    Source     : ST_LogEntry := (Message := 'CopiedData');
    Destination: ST_LogEntry := (Message := '__________'); // Preset dummy
    pSource    : POINTER TO ST_LogEntry;
    pDest      : POINTER TO ST_LogEntry;
    Size       : UDINT;
END_VAR
TEST(__POUNAME());

pSource := ADR(Source);
pDest := ADR(Destination);
Size := SIZEOF(ST_LogEntry);

// Call CopyMemArea
//RingBuffer.CopyMemArea(pDest := pDest, pSource := pSource, Size := Size);

// Assert values match
AssertEquals(
    Actual := Destination.Message,
    Expected := Source.Message,
    Message := 'Expected destination string to match source after memory copy'
);

TEST_FINISHED();
END_METHOD

METHOD PRIVATE GivenEmptyBufferExpectPeekReturnsDefault
VAR
    Peeked         : ST_LogEntry;
	TempString		: STRING := '';
END_VAR
TEST(__POUNAME());

RingBuffer[24].ClearBuffer();
Peeked := RingBuffer[24].PeekObject();

AssertEquals(Actual := Peeked.Message, Expected := TempString, Message := 'Peeked object should be default');
AssertFalse(Condition := RingBuffer[24].RingBufferStatus.ObjectWasPeekedPrimary, Message := 'ObjectPeeked flag should be FALSE when buffer is empty');

TEST_FINISHED();
END_METHOD

METHOD PRIVATE GivenFillBufferExpectIsFullTrue
VAR
    TestObject  : ST_LogEntry := (Message := 'FullTest');
    i           : UDINT;
END_VAR
TEST(__POUNAME());

RingBuffer[25].Initialize();
FOR i := 1 TO RingBuffer[25].RingBufferStatus.BufferCapacity DO
    RingBuffer[25].AddObject(RefObject := TestObject);
END_FOR

AssertTrue(Condition := RingBuffer[25].RingBufferStatus.BufferIsFullPrim, Message := 'Expected BufferIsFullPrim = TRUE');

TEST_FINISHED();
END_METHOD

METHOD PRIVATE GivenFullBufferAddOneExpectOverwriteOldest
VAR
  O1 : ST_LogEntry := (Message := 'A');
  O2 : ST_LogEntry := (Message := 'B');
  O3 : ST_LogEntry := (Message := 'C');
  O4 : ST_LogEntry := (Message := 'D');
  Removed : ST_LogEntry;
END_VAR
TEST(__POUNAME());

RingBuffer[26].Initialize();

// Fill to buffer capacity first
FOR i := gc_test.INDEX_TestFB_RingBuffer_MIN TO UDINT_TO_DINT(RingBuffer[26].P_RingBufferStatus.BufferCapacity) DO
    RingBuffer[26].AddObject(RefObject := O1);
END_FOR

// Add one more to trigger overwrite
RingBuffer[26].AddObject(RefObject := O2);

// Now remove and check FIFO order - first removed should be the overwritten element
RingBuffer[26].RemoveObject(); 
Removed := RingBuffer[26].LastObjRemoved;
AssertEquals(Actual := Removed.Message, Expected := O1.Message, Message := 'Expected first object from overwrite scenario');

TEST_FINISHED();
END_METHOD

METHOD PRIVATE GivenInitExpectDefaultPointerAndState
VAR

	tempValWrite	: PVOID := ADR(RingBuffer[27].Buffer[GPL_RingBuffer.MIN_LOGENTRIES]);
	tempValRemove	: PVOID := ADR(RingBuffer[27].Buffer[GPL_RingBuffer.MIN_LOGENTRIES]);
	tempCount		: UDINT := 0;
END_VAR
TEST(__POUNAME());

// Initialize the RingBuffer
RingBuffer[27].Initialize();

// Assert initial state of pointers and flags
AssertEquals_LWORD(Actual := RingBuffer[27].pWrite, Expected := tempValWrite, Message := 'Expected pWrite at buffer start on init');
AssertEquals_LWORD(Actual := RingBuffer[27].pRemove, Expected := tempValRemove, Message := 'Expected pRemove at buffer start on init');
AssertEquals(Actual := RingBuffer[27].RingBufferStatus.GlobalCounter, Expected := tempCount, Message := 'Expected GlobalCounter to be 0 on init');
AssertFalse(Condition := RingBuffer[27].RingBufferStatus.ObjectWasAddedPrimary, Message := 'Expected ObjectAddedPrimary to be FALSE on init');
AssertFalse(Condition := RingBuffer[27].RingBufferStatus.ObjectWasRemovedPrimary, Message := 'Expected ObjectRemovedPrimary to be FALSE on init');

TEST_FINISHED();
END_METHOD

METHOD PRIVATE GivenLargeStringExpectTruncationOrError
VAR

    TestObject : ST_LogEntry := (Message := 'Hello');
    Removed    : ST_LogEntry;
END_VAR
TEST(__POUNAME());

RingBuffer[28].Initialize();
TestObject.Message := 'ABCDEFGHIJKLMNOPQRSTUVWXYZ';
RingBuffer[28].AddObject(RefObject := TestObject);

AssertTrue(Condition := LEN(RingBuffer[28].Buffer[GPL_RingBuffer.MIN_LOGENTRIES].Message) <= SIZEOF(RingBuffer[28].Buffer[0].Message),
    Message := 'Expected truncation or error for large string');

TEST_FINISHED();
END_METHOD

METHOD PRIVATE GivenMultipleAddInSingleCycleExpectAllStored
VAR

    TestObject : ST_LogEntry := (Message := 'Hello');
    Removed    : ST_LogEntry;
END_VAR
TEST(__POUNAME());

RingBuffer[29].Initialize();
RingBuffer[29].AddObject(RefObject := TestObject);
RingBuffer[29].AddObject(RefObject := TestObject);

AssertEquals_UDINT(Actual := RingBuffer[29].RingBufferStatus.GlobalCounter, Expected := 2,
    Message := 'Expected two objects stored in single cycle');

TEST_FINISHED();
END_METHOD

METHOD PRIVATE GivenMultipleAddsSameCycleExpectAllStored
VAR
  O1 : ST_LogEntry := (Message := 'Alpha');
  O2 : ST_LogEntry := (Message := 'Beta');
END_VAR
TEST(__POUNAME());

RingBuffer[30].Initialize();
RingBuffer[30].AddObject(RefObject := O1);
RingBuffer[30].AddObject(RefObject := O2);

RingBuffer[30].RemoveObject();
AssertEquals(Actual := RingBuffer[30].LastObjRemoved.Message, Expected := O1.Message, Message := 'First object mismatch');

RingBuffer[30].RemoveObject();
AssertEquals(Actual := RingBuffer[30].LastObjRemoved.Message, Expected := O2.Message, Message := 'Second object mismatch');

TEST_FINISHED();
END_METHOD

METHOD PRIVATE GivenMultipleObjectsExpectPeekAlwaysReturnsFirst
VAR
    Peeked			: ST_LogEntry;
	TestObject		: ST_LogEntry;
	TempString1		: STRING := 'First';
	TempString2		: STRING := 'Second';
END_VAR
TEST(__POUNAME());

RingBuffer[31].Initialize();
RingBuffer[31].ClearBuffer();
TestObject.Message	:= TempString1;
RingBuffer[31].AddObject(RefObject := TestObject);
TestObject.Message	:= TempString2;
RingBuffer[31].AddObject(RefObject := TestObject);

Peeked := RingBuffer[31].PeekObject();
AssertEquals(Actual := Peeked.Message, Expected := TempString1, Message := 'Peek should return the first object');

Peeked := RingBuffer[31].PeekObject();
AssertEquals(Actual := Peeked.Message, Expected := TempString1, Message := 'Repeated peek should still return the first object');

TEST_FINISHED();
END_METHOD

METHOD PRIVATE GivenNullRefInputExpectGracefulHandling
VAR

    NullRef    : REFERENCE TO ST_LogEntry;
    InitialCount : UDINT;
END_VAR
TEST(__POUNAME());

RingBuffer[32].Initialize();
// Store initial object count
InitialCount := RingBuffer[32].RingBufferStatus.GlobalCounter;

// Attempt to add a null reference — should not crash or write anything
RingBuffer[32].AddObject(RefObject := NullRef);

// Assert no change in count or flags
AssertEquals(Actual := RingBuffer[32].RingBufferStatus.GlobalCounter, Expected := InitialCount, Message := 'Expected no change in count on null input');
AssertFalse(Condition := RingBuffer[32].RingBufferStatus.ObjectWasAddedPrimary, Message := 'Expected ObjectAddedPrimary to remain FALSE');

TEST_FINISHED();
END_METHOD

METHOD PRIVATE GivenOneObjectAddedExpectPeekReturnsIt
VAR
    TestObj        : ST_LogEntry := (Message := 'Alpha');
    Peeked         : ST_LogEntry;
END_VAR
TEST(__POUNAME());

RingBuffer[33].Initialize();
RingBuffer[33].ClearBuffer();
RingBuffer[33].AddObject(TestObj);
Peeked := RingBuffer[33].PeekObject();

AssertEquals(Actual := Peeked.Message, Expected := TestObj.Message, Message := 'Peeked value should match added object');

TEST_FINISHED();
END_METHOD

METHOD PRIVATE GivenOversizedObject_WhenAdded_ExpectNoAdjacentMemoryCorruption
VAR
    OversizedObject : ST_LogEntry;
    GuardBefore     : DWORD := 16#DEADBEEF;
    GuardAfter      : DWORD := 16#CAFEBABE;
    i               : INT;
    TestString      : STRING(255);
END_VAR
TEST(__POUNAME());

RingBuffer[23].Initialize();

// Create an oversized string (fill to maximum)
FOR i := 1 TO 255 DO
    TestString := CONCAT(TestString, 'X');
END_FOR
OversizedObject.Message := TestString;

// Store guard values to detect memory corruption
GuardBefore := 16#DEADBEEF;
GuardAfter := 16#CAFEBABE;

// Add the oversized object
RingBuffer[23].AddObject(RefObject := OversizedObject);

// Verify guards haven't been corrupted
AssertEquals_DWORD(
    Actual := GuardBefore,
    Expected := 16#DEADBEEF,
    Message := 'Guard before buffer was corrupted'
);

AssertEquals_DWORD(
    Actual := GuardAfter,
    Expected := 16#CAFEBABE,
    Message := 'Guard after buffer was corrupted'
);

// Verify the buffer still functions correctly
RingBuffer[23].RemoveObject();
AssertEquals_UDINT(
    Actual := RingBuffer[23].RingBufferStatus.GlobalCounter,
    Expected := 0,
    Message := 'Buffer should still function after oversized add'
);

TEST_FINISHED();
END_METHOD

METHOD PRIVATE GivenOversizedObjectExpectPartialWriteOrError
VAR
    Oversized   : ST_LogEntry := (Message := 'ABCDEFGHIJKLMNOPQRSTUVWXYZ0123456789ABCDEFGHIJKLMNOPQRSTUVWXYZ0123456789'); // >64 chars
    InitialCount : UDINT;
END_VAR
TEST(__POUNAME());

RingBuffer[34].Initialize();
InitialCount := RingBuffer[34].RingBufferStatus.GlobalCounter;

// Attempt to add an oversized object
RingBuffer[34].AddObject(RefObject := Oversized);

// Validate that no object was added or error was flagged
AssertEquals_UDINT(Actual := RingBuffer[34].RingBufferStatus.GlobalCounter, Expected := InitialCount + 1, Message := 'Expected object to be added');
AssertTrue(Condition := RingBuffer[34].RingBufferStatus.ObjectWasAddedPrimary, Message := 'Expected ObjectAddedPrimary to be TRUE');

TEST_FINISHED();
END_METHOD

METHOD PRIVATE GivenOverwrite_WhenOccurs_ExpectDropCounterIncremented
VAR
    TestObject      : ST_LogEntry;
    i               : UDINT;
    Capacity        : UDINT;
    InitialDrops    : UDINT;
    DropsAfterOverwrite : UDINT;
END_VAR
TEST(__POUNAME());

RingBuffer[60].Initialize();
RingBuffer[60].ClearBuffer();
Capacity := RingBuffer[60].RingBufferStatus.BufferCapacity;

// Note: Check if DropCounter exists in the status structure
// If not, we'll track overwrites via the Overwriting flag

// Fill buffer to capacity
FOR i := 1 TO Capacity DO
    TestObject.Message := CONCAT('Item_', UDINT_TO_STRING(i));
    RingBuffer[60].AddObject(RefObject := TestObject);
END_FOR

// Verify buffer is full
AssertTrue(
    Condition := RingBuffer[60].RingBufferStatus.BufferIsFullPrim,
    Message := 'Buffer should be full before overwrite test'
);

// Store initial state (if DropCounter exists, it would be tracked here)
InitialDrops := 0; // Placeholder - would be actual drop counter if it exists

// Add one more to trigger overwrite
TestObject.Message := 'Overwrite1';
RingBuffer[60].AddObject(RefObject := TestObject);

// Check overwrite occurred
AssertTrue(
    Condition := RingBuffer[60].RingBufferStatus.Overwriting,
    Message := 'Overwriting flag should be TRUE after overwrite'
);

// Add several more overwrites
FOR i := 1 TO 5 DO
    TestObject.Message := CONCAT('Overwrite_', UDINT_TO_STRING(i+1));
    RingBuffer[60].AddObject(RefObject := TestObject);
END_FOR

// Verify buffer still at capacity (not growing)
AssertEquals_UDINT(
    Actual := ULINT_TO_UDINT(RingBuffer[60].RingBufferStatus.ObjectCountInBufferPrim),
    Expected := Capacity,
    Message := 'Buffer count should remain at capacity during overwrites'
);

// Verify we can still read most recent entries
RingBuffer[60].RemoveObject();
// The oldest remaining entry should be one of the overwrite entries
AssertTrue(
    Condition := (LEFT(RingBuffer[60].LastObjRemoved.Message, 9) = 'Overwrite')
                 OR (LEFT(RingBuffer[60].LastObjRemoved.Message, 4) = 'Item'),
    Message := 'Should retrieve valid data after overwrites'
);

// If a drop counter exists, verify it incremented
// DropsAfterOverwrite := <actual drop counter if it exists>
// AssertTrue(
//     Condition := DropsAfterOverwrite > InitialDrops,
//     Message := 'Drop counter should increment on overwrites'
// );

TEST_FINISHED();
END_METHOD

METHOD PRIVATE GivenOverwriteExpectFlagSet
VAR
    TestObject  : ST_LogEntry := (Message := 'OverwriteTest');
    i           : UDINT;
END_VAR
TEST(__POUNAME());

RingBuffer[35].Initialize();
// Fill to capacity
FOR i := 1 TO RingBuffer[35].RingBufferStatus.BufferCapacity DO
    RingBuffer[35].AddObject(RefObject := TestObject);
END_FOR

// This next add should trigger overwrite
RingBuffer[35].AddObject(RefObject := TestObject);
AssertTrue(Condition := RingBuffer[35].RingBufferStatus.Overwriting, Message := 'Expected Overwriting = TRUE');

TEST_FINISHED();
END_METHOD

METHOD PRIVATE GivenOverwriteOccursExpectOnlyRecentN
VAR

    TestObject : ST_LogEntry := (Message := 'Hello');
    Removed    : ST_LogEntry;
END_VAR
TEST(__POUNAME());

RingBuffer[36].Initialize();
FOR i := 1 TO (RingBuffer[36].RingBufferStatus.BufferCapacity + 2) DO
    RingBuffer[36].AddObject(RefObject := TestObject);
END_FOR
AssertEquals_UDINT(
    Actual := ULINT_TO_UDINT(RingBuffer[36].RingBufferStatus.ObjectCountInBufferPrim),
    Expected := RingBuffer[36].RingBufferStatus.BufferCapacity,
    Message := 'Expected buffer to hold only most recent N elements'
);
TEST_FINISHED();
END_METHOD

METHOD PRIVATE GivenOverwriteThenReadExpectMostRecent
VAR
    TestObject 	: ST_LogEntry;
    ReadObj    	: ST_LogEntry;
    Obj1       	: ST_LogEntry;
    Obj2       	: ST_LogEntry;
    Obj3       	: ST_LogEntry;
    Obj4       	: ST_LogEntry;
    Obj5       	: ST_LogEntry;
	Obj6	 	: ST_LogEntry;
	i			: INT;
END_VAR
TEST(__POUNAME());

RingBuffer[37].Initialize();
Obj1.Message := '1';
Obj2.Message := '2';
Obj3.Message := '3';
Obj4.Message := '4';
Obj5.Message := '5';
Obj6.Message := '6';

// Add Obj1
RingBuffer[37].AddObject(RefObject := Obj1);

// Fill buffer to capacity with Obj2, Obj3, etc.
// This will cause Obj1 to be overwritten when we reach capacity + 1
FOR i := 1 TO DINT_TO_INT(UDINT_TO_DINT(RingBuffer[37].RingBufferStatus.BufferCapacity) - 1) DO
	TestObject.Message := CONCAT('Filler', INT_TO_STRING(i));
	RingBuffer[37].AddObject(RefObject := TestObject);
END_FOR

// Add Obj2 - this will overwrite Obj1, making Obj2 the oldest
RingBuffer[37].AddObject(RefObject := Obj2);

// Verify overwriting occurred
AssertTrue(RingBuffer[37].RingBufferStatus.Overwriting, 'Expected overwriting to have occurred');

RingBuffer[37].ReadObject();
ReadObj := RingBuffer[37].LastObjRead;

AssertEquals(Actual := ReadObj.Message, Expected := Obj2.Message,
             Message := 'Expected oldest object (Obj2) after overwrite');

TEST_FINISHED();
END_METHOD

METHOD PRIVATE GivenOverwriteThenRemoveExpectOverwriteCleared
VAR
	DummyObj     : ST_LogEntry;
	i            : INT;
	Capacity     : UDINT;
	ExpectedCountAfterRemove : UDINT;
	ExpectedByteCountAfterRemove : ULINT;
END_VAR
TEST(__POUNAME());

RingBuffer[38].Initialize();
RingBuffer[38].ClearBuffer();

// Get capacity
Capacity := RingBuffer[38].RingBufferStatus.BufferCapacity;

// Fill to capacity + 2 to trigger overwriting
FOR i := 1 TO UDINT_TO_INT(Capacity + 2) DO
    RingBuffer[38].AddObject(RefObject := DummyObj);
END_FOR

AssertTrue(RingBuffer[38].RingBufferStatus.Overwriting, 'Expected overwrite flag set after overfill');
AssertEquals_UDINT(Capacity, RingBuffer[38].RingBufferStatus.GlobalCounter, 'Expected GlobalCounter at capacity after overwrite');

// Remove one object
RingBuffer[38].RemoveObject();

// Calculate expected values after removing one object
ExpectedCountAfterRemove := Capacity - 1;
ExpectedByteCountAfterRemove := UDINT_TO_ULINT(ExpectedCountAfterRemove * SIZEOF(DummyObj));

// Expect overwrite cleared (buffer is no longer full)
AssertFalse(RingBuffer[38].RingBufferStatus.Overwriting, 'Expected Overwriting = FALSE after remove');
AssertFalse(RingBuffer[38].RingBufferStatus.WillOverwrite, 'Expected WillOverwrite = FALSE after remove');
AssertEquals_UDINT(ExpectedCountAfterRemove, RingBuffer[38].RingBufferStatus.GlobalCounter, 'Expected GlobalCounter = capacity - 1');
AssertEquals_ULINT(ExpectedByteCountAfterRemove, RingBuffer[38].RingBufferStatus.ByteCountInBufferPrim, 'Expected ByteCountInBuffer = (capacity-1)*SIZEOF(DummyObj) after remove');

TEST_FINISHED();
END_METHOD

METHOD PRIVATE GivenPeekAndReadExpectFlagsSet
VAR
    TestObject  : ST_LogEntry := (Message := 'PeekReadTest');
END_VAR
TEST(__POUNAME());

RingBuffer[39].Initialize();
RingBuffer[39].AddObject(RefObject := TestObject);

RingBuffer[39].PeekObject();
AssertTrue(Condition := RingBuffer[39].RingBufferStatus.ObjectWasPeekedPrimary, Message := 'Expected ObjectWasPeekedPrimary = TRUE');

RingBuffer[39].ReadObject();
AssertTrue(Condition := RingBuffer[39].RingBufferStatus.ObjectWasReadPrimary, Message := 'Expected ObjectWasReadPrimary = TRUE');

TEST_FINISHED();
END_METHOD

METHOD PRIVATE GivenPeekThenClearPeekedFlagExpectReset
VAR
    TestObject      : ST_LogEntry := (Message := 'PeekTest');
    PeekedObject    : ST_LogEntry;
END_VAR
TEST(__POUNAME());

RingBuffer[40].Initialize();
// Add an object to ensure there's something to peek
RingBuffer[40].AddObject(RefObject := TestObject);

// Perform a peek operation
PeekedObject := RingBuffer[40].PeekObject();

// Ensure the object was peeked correctly
AssertEquals(Actual := PeekedObject.Message, Expected := TestObject.Message, Message := 'Expected Peek to return the correct object');
AssertTrue(Condition := RingBuffer[40].RingBufferStatus.ObjectWasPeekedPrimary, Message := 'Expected ObjectPeeked flag to be set after peek');

// Clear the flag manually or through any provided method
RingBuffer[40].ClearStatusFlagPeeked();

// Ensure the flag was reset
AssertFalse(Condition := RingBuffer[40].RingBufferStatus.ObjectWasPeekedPrimary, Message := 'Expected ObjectPeeked flag to be cleared');

TEST_FINISHED();
END_METHOD

METHOD PRIVATE GivenRapidAddRemoveInLoopExpectCorrectFinalCount

VAR
    TestObject  : ST_LogEntry := (Message := 'RapidIO');
    i           : INT;
    FinalCount  : UDINT;
END_VAR
TEST(__POUNAME());

RingBuffer[41].Initialize();
// Perform rapid add/remove operations in a loop
FOR i := 1 TO 100 DO
    RingBuffer[41].AddObject(RefObject := TestObject);
    RingBuffer[41].RemoveObject();
END_FOR

// After each Add/Remove pair, the buffer should remain empty
FinalCount := RingBuffer[41].RingBufferStatus.GlobalCounter;
AssertEquals_UDINT(Actual := FinalCount, Expected := 0, Message := 'Expected final count to be zero after rapid add/remove loop');

TEST_FINISHED();
END_METHOD

METHOD PRIVATE GivenReadFromEmptyExpectNoCrashOrInvalid
VAR

    TestObject : ST_LogEntry;
    ReadObj    : ST_LogEntry;
    Obj1       : ST_LogEntry;
    Obj2       : ST_LogEntry;
    Obj3       : ST_LogEntry;
    Obj4       : ST_LogEntry;
END_VAR
TEST(__POUNAME());

RingBuffer[42].ClearBuffer();
RingBuffer[42].ReadObject();

AssertFalse(Condition := RingBuffer[42].RingBufferStatus.ObjectWasReadPrimary,
            Message := 'Expected no object to be read from empty buffer');
			
TEST_FINISHED();
END_METHOD

METHOD PRIVATE GivenReadThenClearStatusExpectFlagsReset
VAR
    TestObject  : ST_LogEntry := (Message := 'StatusCheck');
    TempObj     : ST_LogEntry;
    StatusBefore, StatusAfter : BOOL;
END_VAR
TEST(__POUNAME());

RingBuffer[43].Initialize();
// Add and read to set the status flag
RingBuffer[43].AddObject(RefObject := TestObject);
TempObj := RingBuffer[43].ReadObject();

// Verify the read status flag is set
StatusBefore := RingBuffer[43].RingBufferStatus.ObjectWasReadPrimary;
AssertTrue(Condition := StatusBefore, Message := 'Expected ObjectRead flag to be TRUE after read');

// Now clear the status
RingBuffer[43].ClearStatusFlagAdded();
RingBuffer[43].ClearStatusFlagPeeked();
RingBuffer[43].ClearStatusFlagRead();
RingBuffer[43].ClearStatusFlagRemoved();

// Verify the status flag is reset
StatusAfter := RingBuffer[43].RingBufferStatus.ObjectWasReadPrimary;
AssertFalse(Condition := StatusAfter, Message := 'Expected ObjectRead flag to be FALSE after ClearStatusFlags');

TEST_FINISHED();
END_METHOD

METHOD PRIVATE GivenReadThenRemoveExpectCorrectFlagsAndCounts
VAR
	DummyObj     : ST_LogEntry;
	i            : INT;
	ReadObj      : ST_LogEntry;
	testval1	: UDINT := 1;
	testval2	: UDINT := 2;
END_VAR
TEST(__POUNAME());

RingBuffer[44].Initialize();
RingBuffer[44].ClearBuffer();

// Add 3 objects
FOR i := 1 TO 3 DO
	RingBuffer[44].AddObject(RefObject := DummyObj);
END_FOR

// Read
ReadObj := RingBuffer[44].ReadObject();
AssertTrue(RingBuffer[44].RingBufferStatus.ObjectWasReadPrimary, 'Expected ObjectWasReadPrimary = TRUE');
AssertEquals(testval2, RingBuffer[44].RingBufferStatus.GlobalCounter, 'Expected GlobalCounter after read = 2');

// Remove
RingBuffer[44].RemoveObject();
AssertTrue(RingBuffer[44].RingBufferStatus.ObjectWasRemovedPrimary, 'Expected ObjectWasRemovedPrimary = TRUE');
AssertEquals(testval1, RingBuffer[44].RingBufferStatus.GlobalCounter, 'Expected GlobalCounter after remove = 1');

TEST_FINISHED();
END_METHOD

METHOD PRIVATE GivenRemoveBeyondCapacity_ExpectSafeReset
VAR
    TestObject      : ST_LogEntry := (Message := 'TestData');
    i               : UDINT;
    Capacity        : UDINT;
    RemoveError     : BOOL;
    ExpectedString  : STRING := 'AfterExcess';
END_VAR
TEST(__POUNAME());

RingBuffer[59].Initialize();
RingBuffer[59].ClearBuffer();
Capacity := RingBuffer[59].RingBufferStatus.BufferCapacity;

// Test 1: Remove from empty buffer multiple times
FOR i := 1 TO 10 DO
    RingBuffer[59].RemoveObject();
END_FOR

// Buffer should remain stable
AssertEquals_UDINT(
    Actual := RingBuffer[59].RingBufferStatus.GlobalCounter,
    Expected := 0,
    Message := 'Counter should remain 0 after multiple removes from empty'
);

AssertFalse(
    Condition := RingBuffer[59].RingBufferStatus.ObjectWasRemovedPrimary,
    Message := 'Remove flag should be FALSE when removing from empty'
);

// Test 2: Add some items
FOR i := 1 TO 3 DO
    RingBuffer[59].AddObject(RefObject := TestObject);
END_FOR

// Test 3: Remove more than what's available
FOR i := 1 TO 10 DO
    RingBuffer[59].RemoveObject();
END_FOR

AssertEquals_UDINT(
    Actual := RingBuffer[59].RingBufferStatus.GlobalCounter,
    Expected := 0,
    Message := 'Counter should be 0 after excess removes'
);

// Test 4: Verify buffer still works after excess removes
TestObject.Message := ExpectedString;
RingBuffer[59].AddObject(RefObject := TestObject);

AssertEquals_UDINT(
    Actual := RingBuffer[59].RingBufferStatus.GlobalCounter,
    Expected := 1,
    Message := 'Buffer should still accept adds after excess removes'
);

RingBuffer[59].RemoveObject();
AssertEquals(
    Actual := RingBuffer[59].LastObjRemoved.Message,
    Expected := ExpectedString,
    Message := 'Should retrieve correct data after excess removes'
);

// Test 5: Stress test - many excess removes
FOR i := 1 TO 1000 DO
    RingBuffer[59].RemoveObject();
END_FOR

// Verify pointers haven't wrapped incorrectly
AssertEquals_UDINT(
    Actual := RingBuffer[59].RingBufferStatus.GlobalCounter,
    Expected := 0,
    Message := 'Counter stable after 1000 excess removes'
);

TEST_FINISHED();
END_METHOD

METHOD PRIVATE GivenRemoveFromEmptyExpectError
VAR
  Error : BOOL;
END_VAR
TEST(__POUNAME());

RingBuffer[47].Initialize();
RingBuffer[47].RemoveObject();
Error := RingBuffer[47].RingBufferStatus.ObjectWasRemovedPrimary = FALSE;

AssertTrue(Condition := Error, Message := 'Expected error when removing from empty buffer');

TEST_FINISHED();
END_METHOD

METHOD PRIVATE GivenRemoveObjectExpectLastRemovedMatchesExpected
VAR

    Obj1       : ST_LogEntry := (Message := 'ItemOne');
    Obj2       : ST_LogEntry := (Message := 'ItemTwo');
    Removed    : ST_LogEntry;
END_VAR
TEST(__POUNAME());

RingBuffer[46].Initialize();
// Add two items to the buffer
RingBuffer[46].AddObject(RefObject := Obj1);
RingBuffer[46].AddObject(RefObject := Obj2);

// Remove the first item and check if LastObjRemoved is set correctly
RingBuffer[46].RemoveObject();
Removed := RingBuffer[46].LastObjRemoved;
AssertEquals(Actual := Removed.Message, Expected := Obj1.Message, Message := 'Expected first removed object to be Obj1');

// Remove the second item and check again
RingBuffer[46].RemoveObject();
Removed := RingBuffer[46].LastObjRemoved;
AssertEquals(Actual := Removed.Message, Expected := Obj2.Message, Message := 'Expected second removed object to be Obj2');

TEST_FINISHED();
END_METHOD

METHOD PRIVATE GivenRemoveOnEmptyExpectNoCrash
VAR
    TestObject : ST_LogEntry := (Message := 'Hello');
    Removed    : ST_LogEntry;
    Error       : BOOL;
END_VAR
TEST(__POUNAME());

RingBuffer[49].Initialize();
RingBuffer[49].RemoveObject();
Error := RingBuffer[49].RingBufferStatus.ObjectWasRemovedPrimary = FALSE;
AssertTrue(Condition := Error, Message := 'Expected error when removing from empty buffer');

TEST_FINISHED();
END_METHOD

METHOD PRIVATE GivenRemovePointerWrapsAroundExpectValidRead
VAR
    TestObject  : ST_LogEntry := (Message := 'WrapTest');
    Removed     : ST_LogEntry;
    i           : UDINT;
	teststring	: STRING(GPL_RingBuffer.STRING_LENGTH);
END_VAR
TEST(__POUNAME());

RingBuffer[50].Initialize();
FOR i := 1 TO RingBuffer[50].RingBufferStatus.BufferCapacity DO
    TestObject.Message := CONCAT('Val_', DINT_TO_STRING(i));
    RingBuffer[50].AddObject(RefObject := TestObject);
    RingBuffer[50].RemoveObject();
END_FOR

// Force wraparound
teststring	:= 'WrapVal';
TestObject.Message := teststring;
RingBuffer[50].AddObject(RefObject := TestObject);
RingBuffer[50].RemoveObject();

Removed := RingBuffer[50].LastObjRemoved;

AssertEquals(
    Actual := Removed.Message,
    Expected := teststring,
    Message := 'Expected correct object after remove pointer wraparound'
);

TEST_FINISHED();
END_METHOD

METHOD PRIVATE GivenRemoveThenReadExpectNoNewData
VAR

    TestObject : ST_LogEntry;
    ReadObj    : ST_LogEntry;
    Obj1       : ST_LogEntry;
    Obj2       : ST_LogEntry;
    Obj3       : ST_LogEntry;
    Obj4       : ST_LogEntry;
END_VAR
TEST(__POUNAME());

RingBuffer[51].Initialize();
TestObject.Message := 'Alpha';
RingBuffer[51].AddObject(RefObject := TestObject);
RingBuffer[51].RemoveObject();
RingBuffer[51].ReadObject();

AssertFalse(Condition := RingBuffer[51].RingBufferStatus.ObjectWasReadPrimary,
            Message := 'Expected no valid object after remove');
			
TEST_FINISHED();
END_METHOD

METHOD PRIVATE GivenUpdateRemovePointerBoundaryExpectCorrectWrap
VAR
    TestObject      : ST_LogEntry := (Message := 'WrapTest');
    PointerBefore   : PVOID;
    PointerAfter    : PVOID;
    DidWrap         : BOOL;
    i               : UDINT;
	ExpectedIndex	: ULINT;
END_VAR
TEST(__POUNAME());

RingBuffer[52].Initialize();
FOR i := 1 TO RingBuffer[52].RingBufferStatus.BufferCapacity DO
    RingBuffer[52].AddObject(RefObject := TestObject);
END_FOR

FOR i := 1 TO RingBuffer[52].RingBufferStatus.BufferCapacity DO
    RingBuffer[52].RemoveObject();
END_FOR

// Perform one more Add and Remove
RingBuffer[52].AddObject(RefObject := TestObject);
RingBuffer[52].RemoveObject();

// Now calculate what the RemoveIndex *should* be
ExpectedIndex := (RingBuffer[52].RemoveIncrement MOD RingBuffer[52].RingBufferStatus.BufferCapacity)
                 + GPL_RingBuffer.MIN_LOGENTRIES;

// Compare with actual value in FB
AssertEquals_UDINT(
    Actual := ULINT_TO_UDINT(RingBuffer[52].RemoveIndex),
    Expected := ULINT_TO_UDINT(ExpectedIndex),
    Message := 'Expected RemoveIndex to advance correctly (wrap around if at boundary)'
);

TEST_FINISHED();
END_METHOD

METHOD PRIVATE GivenUpdateWritePointerBoundaryExpectCorrectWrap
VAR
    TestObject   : ST_LogEntry := (Message := 'WrapTest');
    i            : DINT;
    InitialIndex : UDINT;
    FinalIndex   : UDINT;
END_VAR
TEST(__POUNAME());

// Assume buffer capacity is N, writing N+1 elements should wrap the pointer
InitialIndex := RingBuffer[53].WriteIndex;
FOR i := 1 TO (RingBuffer[53].RingBufferStatus.BufferCapacity + 1) DO
    RingBuffer[53].AddObject(RefObject := TestObject);
END_FOR
FinalIndex := RingBuffer[53].WriteIndex;

// Final write index should have wrapped around to (Initial + 1) mod Capacity
AssertEquals_UDINT(
    Actual := FinalIndex, 
    Expected := (InitialIndex + 1) MOD RingBuffer[53].RingBufferStatus.BufferCapacity,
    Message := 'Expected write pointer to wrap around after full buffer write');

TEST_FINISHED();
END_METHOD

METHOD PRIVATE GivenWrapAroundManyTimes_ExpectCountersStable
VAR
    TestObject      : ST_LogEntry;
    i, j            : UDINT;
    Capacity        : UDINT;
    NumWraps        : UDINT := 100; // Number of times to wrap around
    ExpectedCount   : UDINT;
    InitialWriteIdx : UDINT;
    InitialRemoveIdx: UDINT;
    Removed         : ST_LogEntry;
    ExpectedMessage1: STRING(80);
    ExpectedMessage2: STRING := 'FinalTest';
END_VAR
TEST(__POUNAME());

RingBuffer[61].Initialize();
RingBuffer[61].ClearBuffer();
Capacity := RingBuffer[61].RingBufferStatus.BufferCapacity;

// Test 1: Many wrap-arounds with add/remove pattern
FOR j := 1 TO NumWraps DO
    // Fill buffer completely
    FOR i := 1 TO Capacity DO
        TestObject.Message := CONCAT('Wrap', CONCAT(UDINT_TO_STRING(j), CONCAT('_Item', UDINT_TO_STRING(i))));
        RingBuffer[61].AddObject(RefObject := TestObject);
    END_FOR

    // Remove all items
    FOR i := 1 TO Capacity DO
        RingBuffer[61].RemoveObject();
    END_FOR

    // Verify buffer is empty after each cycle
    AssertEquals_UDINT(
        Actual := RingBuffer[61].RingBufferStatus.GlobalCounter,
        Expected := 0,
        Message := CONCAT('Buffer should be empty after wrap cycle ', UDINT_TO_STRING(j))
    );
END_FOR

// Test 2: Continuous overwrites for many cycles
RingBuffer[61].ClearBuffer();
FOR i := 1 TO (Capacity * NumWraps) DO
    TestObject.Message := CONCAT('Continuous_', UDINT_TO_STRING(i));
    RingBuffer[61].AddObject(RefObject := TestObject);
END_FOR

// Should only have last 'Capacity' items
AssertEquals_UDINT(
    Actual := ULINT_TO_UDINT(RingBuffer[61].RingBufferStatus.ObjectCountInBufferPrim),
    Expected := Capacity,
    Message := 'Buffer should contain exactly capacity items after many overwrites'
);

// Test 3: Verify FIFO order still maintained after many wraps
ExpectedCount := (Capacity * NumWraps) - Capacity + 1; // First item that should be in buffer
ExpectedMessage1 := CONCAT('Continuous_', UDINT_TO_STRING(ExpectedCount));
RingBuffer[61].RemoveObject();
Removed := RingBuffer[61].LastObjRemoved;
AssertEquals(
    Actual := Removed.Message,
    Expected := ExpectedMessage1,
    Message := 'FIFO order should be maintained after many wrap-arounds'
);

// Test 4: Stress test with alternating patterns
RingBuffer[61].ClearBuffer();
FOR j := 1 TO 1000 DO
    // Add 3, remove 2 pattern
    FOR i := 1 TO 3 DO
        TestObject.Message := CONCAT('Stress_', UDINT_TO_STRING(j * 3 + i));
        RingBuffer[61].AddObject(RefObject := TestObject);
    END_FOR

    IF RingBuffer[61].RingBufferStatus.GlobalCounter >= 2 THEN
        RingBuffer[61].RemoveObject();
        RingBuffer[61].RemoveObject();
    END_IF
END_FOR

// Verify counters are still consistent
AssertTrue(
    Condition := RingBuffer[61].RingBufferStatus.GlobalCounter <= Capacity,
    Message := 'Global counter should not exceed capacity'
);

AssertEquals_ULINT(
    Actual := RingBuffer[61].RingBufferStatus.ByteCountInBufferPrim,
    Expected := RingBuffer[61].RingBufferStatus.ObjectCountInBufferPrim * SIZEOF(TestObject),
    Message := 'Byte count should match object count * size after stress test'
);

// Test 5: Verify buffer still functional after stress
RingBuffer[61].ClearBuffer();

// Verify buffer is actually empty after clear
AssertEquals_UDINT(
    Actual := RingBuffer[61].RingBufferStatus.GlobalCounter,
    Expected := 0,
    Message := 'Buffer should be empty after ClearBuffer'
);

TestObject.Message := ExpectedMessage2;
RingBuffer[61].AddObject(RefObject := TestObject);

// Verify object was added
AssertEquals_UDINT(
    Actual := RingBuffer[61].RingBufferStatus.GlobalCounter,
    Expected := 1,
    Message := 'Buffer should contain 1 object after add'
);

RingBuffer[61].RemoveObject();
AssertEquals(
    Actual := RingBuffer[61].LastObjRemoved.Message,
    Expected := ExpectedMessage2,
    Message := 'Buffer should still function correctly after stress test'
);

TEST_FINISHED();
END_METHOD

METHOD PRIVATE GivenWrapAroundReadPointerExpectCorrectRead
VAR

    TestObject : ST_LogEntry;
    ReadObj    : ST_LogEntry;
    Obj1       : ST_LogEntry;
    Obj2       : ST_LogEntry;
    Obj3       : ST_LogEntry;
    Obj4       : ST_LogEntry;
END_VAR
TEST(__POUNAME());

RingBuffer[54].Initialize();
Obj1.Message := 'First';
Obj2.Message := 'Second';
RingBuffer[54].AddObject(RefObject := Obj1);
RingBuffer[54].AddObject(RefObject := Obj2);
RingBuffer[54].RemoveObject();
RingBuffer[54].RemoveObject();
// Buffer is empty now; add again to force wrap
RingBuffer[54].AddObject(RefObject := Obj2);
RingBuffer[54].ReadObject();
ReadObj := RingBuffer[54].LastObjRead;
AssertEquals(Actual := ReadObj.Message, Expected := Obj2.Message,
             Message := 'Expected correct wraparound read');
			 
TEST_FINISHED();
END_METHOD

METHOD PRIVATE GivenWrapAroundWriteExpectValidRead
VAR

    TestObject : ST_LogEntry := (Message := 'Hello');
    Removed    : ST_LogEntry;
END_VAR
TEST(__POUNAME());
RingBuffer[55].Initialize();
FOR i := 1 TO RingBuffer[55].RingBufferStatus.BufferCapacity DO
    RingBuffer[55].AddObject(RefObject := TestObject);
END_FOR
RingBuffer[55].RemoveObject(); Removed := RingBuffer[55].LastObjRemoved;
AssertEquals(Actual := Removed.Message, Expected := TestObject.Message,
    Message := 'Expected matching string after wrap-around');
TEST_FINISHED();
END_METHOD

METHOD PRIVATE GivenWritePointerWrapsAroundExpectValidOverwrite
VAR

    Obj1       : ST_LogEntry := (Message := 'First');
    Obj2       : ST_LogEntry := (Message := 'Second');
    Obj3       : ST_LogEntry := (Message := 'Third');
    Obj4       : ST_LogEntry := (Message := 'Fourth');
    Removed    : ST_LogEntry;
    Capacity   : UDINT;
END_VAR
TEST(__POUNAME());

RingBuffer[56].Initialize();
// Get capacity from RingBuffer
Capacity := RingBuffer[56].RingBufferStatus.BufferCapacity;

// Fill the buffer exactly to capacity
RingBuffer[56].AddObject(RefObject := Obj1);
RingBuffer[56].AddObject(RefObject := Obj2);
RingBuffer[56].AddObject(RefObject := Obj3);

// Remove one object to make room and cause wrap-around on next add
RingBuffer[56].RemoveObject(); // Removes Obj1

// Add another object, which should go to the start (wrap-around)
RingBuffer[56].AddObject(RefObject := Obj4);

// Remove remaining to confirm order and correct overwrite
RingBuffer[56].RemoveObject(); Removed := RingBuffer[56].LastObjRemoved;
AssertEquals(Actual := Removed.Message, Expected := Obj2.Message, Message := 'Expected Second');

RingBuffer[56].RemoveObject(); Removed := RingBuffer[56].LastObjRemoved;
AssertEquals(Actual := Removed.Message, Expected := Obj3.Message, Message := 'Expected Third');

RingBuffer[56].RemoveObject(); Removed := RingBuffer[56].LastObjRemoved;
AssertEquals(Actual := Removed.Message, Expected := Obj4.Message, Message := 'Expected Fourth after wrap-around write');

TEST_FINISHED();
END_METHOD

METHOD PRIVATE GivenZeroCapacityBufferExpectNoWrite
VAR

    Obj        : ST_LogEntry := (Message := 'ShouldNotWrite');
    WasWritten : BOOL;
END_VAR
TEST(__POUNAME());

RingBuffer[57].Initialize();

// Normal buffer should work
RingBuffer[57].AddObject(RefObject := Obj);

// Evaluate if it was written — check Add flag
WasWritten := RingBuffer[57].RingBufferStatus.ObjectWasAddedPrimary;

// Assert that object was added
AssertTrue(Condition := WasWritten, Message := 'Expected object to be written to buffer');

TEST_FINISHED();
END_METHOD

METHOD PRIVATE Test_BufferStatus_Add4Remove2
VAR
    DummyObj      : ST_LogEntry; // Replace with actual type
    i             : INT;
    Capacity      : UDINT;
    After4        : UDINT;
    After2        : UDINT;
    AtCapacity    : UDINT;
    BytesAfter4   : ULINT;
    BytesAfter2   : ULINT;
    BytesAtCapacity : ULINT;
END_VAR
TEST(__POUNAME());

// Arrange: Start with empty state
RingBuffer[45].Initialize();
RingBuffer[45].ClearBuffer();
Capacity := RingBuffer[45].RingBufferStatus.BufferCapacity;

// Act: Add 4 objects
FOR i := 1 TO 4 DO
    RingBuffer[45].AddObject(RefObject := DummyObj);
END_FOR

// Assert after Add 4
After4 := 4;
BytesAfter4 := UDINT_TO_ULINT(After4 * SIZEOF(DummyObj));
AssertEquals_UDINT(Expected := After4, Actual := RingBuffer[45].RingBufferStatus.GlobalCounter, Message := 'After Add4: GlobalCounter incorrect');
AssertEquals_ULINT(Expected := BytesAfter4, Actual := RingBuffer[45].RingBufferStatus.ByteCountInBufferPrim, Message := 'After Add4: ByteCountInBuffer incorrect');
AssertFalse(Condition := RingBuffer[45].RingBufferStatus.Overwriting, Message := 'After Add4: Overwriting should be FALSE');
AssertFalse(Condition := RingBuffer[45].RingBufferStatus.WillOverwrite, Message := 'After Add4: WillOverwrite should be FALSE');

// Act: Remove 2 objects
FOR i := 1 TO 2 DO
    RingBuffer[45].RemoveObject();
END_FOR

// Assert after Remove 2
After2 := 2;
BytesAfter2 := UDINT_TO_ULINT(After2 * SIZEOF(DummyObj));
AssertEquals_UDINT(Expected := After2, Actual := RingBuffer[45].RingBufferStatus.GlobalCounter, Message := 'After Remove2: GlobalCounter should be 2');
AssertEquals_ULINT(Expected := BytesAfter2, Actual := RingBuffer[45].RingBufferStatus.ByteCountInBufferPrim, Message := 'After Remove2: ByteCountInBuffer should reflect 2 objects');
AssertFalse(Condition := RingBuffer[45].RingBufferStatus.Overwriting, Message := 'After Remove2: Overwriting should be FALSE');
AssertFalse(Condition := RingBuffer[45].RingBufferStatus.WillOverwrite, Message := 'After Remove2: WillOverwrite should be FALSE');

// Act: Add enough objects to reach capacity (capacity - 2 more objects)
FOR i := 1 TO UDINT_TO_INT(Capacity - After2) DO
    RingBuffer[45].AddObject(RefObject := DummyObj);
END_FOR

// Assert after reaching capacity
AtCapacity := Capacity;
BytesAtCapacity := UDINT_TO_ULINT(AtCapacity * SIZEOF(DummyObj));
AssertEquals_UDINT(Expected := AtCapacity, Actual := RingBuffer[45].RingBufferStatus.GlobalCounter, Message := 'After reaching capacity: GlobalCounter should equal capacity');
AssertEquals_ULINT(Expected := BytesAtCapacity, Actual := RingBuffer[45].RingBufferStatus.ByteCountInBufferPrim, Message := 'After reaching capacity: ByteCountInBuffer should reflect capacity objects');
AssertFalse(Condition := RingBuffer[45].RingBufferStatus.Overwriting, Message := 'After reaching capacity: Overwriting should be FALSE (no overwrite yet)');
AssertTrue(Condition := RingBuffer[45].RingBufferStatus.WillOverwrite, Message := 'After reaching capacity: WillOverwrite should be TRUE (next add will overwrite)');

TEST_FINISHED();
END_METHOD

METHOD PRIVATE Test_BufferStatus_AfterAddAndRemove
VAR
    DummyObj     : ST_LogEntry; // Replace with actual type
    i            : INT;
    Capacity     : UDINT;
    After2       : UDINT;
    BytesAfter2  : ULINT;
    AfterOverwrite : UDINT;
    BytesAfterOverwrite : ULINT;
    AfterRemove  : UDINT;
    BytesAfterRemove : ULINT;
END_VAR
TEST(__POUNAME());
// Arrange
RingBuffer[48].Initialize();
RingBuffer[48].ClearBuffer(); // Reset state
Capacity := RingBuffer[48].RingBufferStatus.BufferCapacity;

// Act: Add 2 objects
FOR i := 1 TO 2 DO
    RingBuffer[48].AddObject(RefObject := DummyObj);
END_FOR

// Assert after 2 adds
After2 := 2;
BytesAfter2 := UDINT_TO_ULINT(After2 * SIZEOF(DummyObj));
AssertEquals_UDINT(Expected := After2, Actual := RingBuffer[48].RingBufferStatus.GlobalCounter, Message := 'After Add2: GlobalCounter incorrect');
AssertEquals_ULINT(Expected := BytesAfter2, Actual := RingBuffer[48].RingBufferStatus.ByteCountInBufferPrim, Message := 'After Add2: ByteCountInBuffer incorrect');
AssertFalse(Condition := RingBuffer[48].RingBufferStatus.Overwriting, Message := 'After Add2: Overwriting should be FALSE');
AssertFalse(Condition := RingBuffer[48].RingBufferStatus.WillOverwrite, Message := 'After Add2: WillOverwrite should be FALSE');

// Act: Add (Capacity + 5) more objects to trigger overwriting
// This will: fill buffer to capacity, then overwrite 5 entries
FOR i := 1 TO UDINT_TO_INT(Capacity + 5 - After2) DO
    RingBuffer[48].AddObject(RefObject := DummyObj);
END_FOR

// Assert after overwrites (total attempted = Capacity + 5, but buffer holds Capacity)
AfterOverwrite := Capacity;
BytesAfterOverwrite := UDINT_TO_ULINT(AfterOverwrite * SIZEOF(DummyObj));
AssertEquals_UDINT(Expected := AfterOverwrite, Actual := RingBuffer[48].RingBufferStatus.GlobalCounter, Message := 'After overwriting: GlobalCounter should be capped at capacity');
AssertEquals_ULINT(Expected := BytesAfterOverwrite, Actual := RingBuffer[48].RingBufferStatus.ByteCountInBufferPrim, Message := 'After overwriting: ByteCountInBuffer should reflect capacity objects');
AssertTrue(Condition := RingBuffer[48].RingBufferStatus.Overwriting, Message := 'After overwriting: Overwriting should be TRUE (overwrite occurred)');
AssertTrue(Condition := RingBuffer[48].RingBufferStatus.WillOverwrite, Message := 'After overwriting: WillOverwrite should be TRUE (still full)');

// Act: Remove 1 object
RingBuffer[48].RemoveObject();

// Assert after Remove 1
AfterRemove := Capacity - 1;
BytesAfterRemove := UDINT_TO_ULINT(AfterRemove * SIZEOF(DummyObj));
AssertEquals_UDINT(Expected := AfterRemove, Actual := RingBuffer[48].RingBufferStatus.GlobalCounter, Message := 'After Remove: GlobalCounter should be capacity - 1');
AssertEquals_ULINT(Expected := BytesAfterRemove, Actual := RingBuffer[48].RingBufferStatus.ByteCountInBufferPrim, Message := 'After Remove: ByteCountInBuffer incorrect');
AssertFalse(Condition := RingBuffer[48].RingBufferStatus.Overwriting, Message := 'After Remove: Overwriting should be FALSE');
AssertFalse(Condition := RingBuffer[48].RingBufferStatus.WillOverwrite, Message := 'After Remove: WillOverwrite should be FALSE');

TEST_FINISHED();
END_METHOD

END_FUNCTION_BLOCK

// RingBuffer/POUs/FB_RingBufferLogEntry
{attribute 'no_explicit_call' := 'do not call this POU directly'}
FUNCTION_BLOCK FB_RingBufferLogEntry EXTENDS FB_RingBufferBase IMPLEMENTS I_RingBufferLogEntry
VAR
  Buffer              	: ARRAY[GPL_RingBuffer.MIN_LOGENTRIES..GPL_RingBuffer.MAX_LOGENTRIES] 
                        	OF ST_LogEntry;
  LastObjRemoved		: ST_LogEntry;
  LastObjPeeked			: ST_LogEntry;
  LastObjRead			: ST_LogEntry;
END_VAR

METHOD PUBLIC AddObject
VAR_INPUT
    RefObject : REFERENCE TO ST_LogEntry;
END_VAR
VAR_OUTPUT
    Error : BOOL;
END_VAR
VAR
    ByteSize   : UDINT;
    ByteOffset : UDINT;
    WriteAddr  : PVOID;
END_VAR
Error := FALSE;
ByteSize := RingBufferConfiguration.ByteCountOfDataObj;

(* ---------- GUARDS ---------- *)
IF (RingBufferStatus.BufferCapacity = 0) OR (NOT __ISVALIDREF(RefObject)) THEN
    Error := TRUE;                           (* zero-capacity or bogus ref *)
    IF BaseConfiguration.LogTraceConfiguration.What.xLogToEventLogger THEN
        ADSLOGSTR(
            msgCtrlMask := ADSLOG_MSGTYPE_ERROR,
            msgFmtStr := 'RingBufferLogEntry.AddObject: Invalid buffer capacity or reference',
            strArg := ''
        );
    END_IF
    RETURN;
END_IF;
IF LEN(RefObject.Message) > SIZEOF(RefObject.Message) THEN
    Error := TRUE;                           (* over-sized payload *)
    IF BaseConfiguration.LogTraceConfiguration.What.xLogToEventLogger THEN
        ADSLOGSTR(
            msgCtrlMask := ADSLOG_MSGTYPE_ERROR,
            msgFmtStr := 'RingBufferLogEntry.AddObject: Message too large: %s',
            strArg := RefObject.Message
        );
    END_IF
    RETURN;
END_IF;

(* ---------- PREDICT / PREP ---------- *)
RingBufferStatus.WillOverwrite :=
    (RingBufferStatus.ObjectCountInBufferPrim >= RingBufferStatus.BufferCapacity);

ByteOffset := (WriteIncrement MOD RingBufferStatus.BufferCapacity) * ByteSize;
WriteAddr  := pBufferStart + ByteOffset;

(* ---------- WRITE ---------- *)
RefObject.systimestamp := Tc2_System.F_GetSystemTime();
IF Tc2_System.MEMMOVE(srcAddr := ADR(RefObject), destAddr := WriteAddr, n := ByteSize) <> ByteSize THEN
    Error := TRUE;
    RETURN;
END_IF;

(* ---------- ADVANCE WRITE POINTERS ---------- *)
WriteIncrement := WriteIncrement + 1;
WriteIndex := (WriteIncrement MOD RingBufferStatus.BufferCapacity)
            + GPL_RingBuffer.MIN_LOGENTRIES;

(* ---------- COUNTERS & FLAGS ---------- *)
IF RingBufferStatus.WillOverwrite THEN
    (* buffer is full – push remove side forward one slot *)
    RemoveIncrement := RemoveIncrement + 1;
    pRemove := pBufferStart
             + (RemoveIncrement MOD RingBufferStatus.BufferCapacity) * ByteSize;
    RingBufferStatus.Overwriting := TRUE;              (* occurred *this* cycle *)
    IF BaseConfiguration.LogTraceConfiguration.What.xLogToEventLogger THEN
        ADSLOGSTR(
            msgCtrlMask := ADSLOG_MSGTYPE_WARN,
            msgFmtStr := 'RingBufferLogEntry: Buffer overflow, oldest entry overwritten. Buffer count: %s',
            strArg := UDINT_TO_STRING(RingBufferStatus.ObjectCountInBufferPrim)
        );
    END_IF
ELSE
    RingBufferStatus.ObjectCountInBufferPrim := RingBufferStatus.ObjectCountInBufferPrim + 1;
    RingBufferStatus.GlobalCounter           := RingBufferStatus.GlobalCounter + 1;
    RingBufferStatus.Overwriting             := FALSE;
END_IF;

RingBufferStatus.ObjectWasAddedPrimary := TRUE;

(* ---------- STATE FOR NEXT SCAN ---------- *)
RingBufferStatus.WillOverwrite :=
    (RingBufferStatus.ObjectCountInBufferPrim >= RingBufferStatus.BufferCapacity);

(* ---------- DERIVED VALUES ---------- *)
RingBufferStatus.BufferIsFullPrim :=
    (RingBufferStatus.ObjectCountInBufferPrim = RingBufferStatus.BufferCapacity);
RingBufferStatus.ByteCountInBufferPrim :=
    RingBufferStatus.ObjectCountInBufferPrim * ByteSize;
END_METHOD

METHOD ClearLastRemoved
MEMSET(destAddr := ADR(LastObjRemoved), fillByte := 16#00, n := RingBufferConfiguration.ByteCountOfDataObj);
END_METHOD

PROPERTY P_LastObjectPeeked : REFERENCE TO ST_LogEntry
GET
P_LastObjectPeeked REF= LastObjPeeked;
END_GET
END_PROPERTY

PROPERTY P_LastObjectRead : REFERENCE TO ST_LogEntry
GET
P_LastObjectRead REF= LastObjRead;
END_GET
END_PROPERTY

PROPERTY P_LastObjectRemoved : REFERENCE TO ST_LogEntry
GET
P_LastObjectRemoved REF= LastObjRemoved;
END_GET
END_PROPERTY

PROPERTY P_RingBufferStatus : REFERENCE TO ST_RingBufferStatus
GET
P_RingBufferStatus REF= SUPER^.RingBufferStatus;
END_GET
END_PROPERTY

METHOD PUBLIC PeekObject : ST_LogEntry
PeekIndex := (RemoveIncrement MOD SUPER^.RingBufferStatus.BufferCapacity) + GPL_RingBuffer.MIN_LOGENTRIES;
PeekAddr := pBufferStart + (PeekIndex - GPL_RingBuffer.MIN_LOGENTRIES) * RingBufferConfiguration.ByteCountOfDataObj;

// Step 2: Conditional peek (non-mutating)
IF SUPER^.RingBufferStatus.GlobalCounter > 0 THEN
    SUPER^.RingBufferStatus.CountBytesPeeked := Tc2_System.MEMMOVE(
        srcAddr := PeekAddr,
        destAddr := ADR(LastObjPeeked),
        n := RingBufferConfiguration.ByteCountOfDataObj
    );

    IF SUPER^.RingBufferStatus.CountBytesPeeked > 0 THEN
        RingBufferStatus.ObjectWasPeekedPrimary := TRUE;
		PeekObject	:= LastObjPeeked;
    END_IF
ELSE
    RingBufferStatus.ObjectWasPeekedPrimary := FALSE;
    LastObjPeeked.Message := '';
END_IF
END_METHOD

METHOD ReadObject : ST_LogEntry
VAR_OUTPUT
  Error : BOOL;
END_VAR
// Step 1: Check if buffer has data
IF SUPER^.RingBufferStatus.GlobalCounter > 0 THEN

    // Step 2: Calculate read offset and pointer
    RingBufferConfiguration.ReadByteOffset := (RemoveIncrement MOD RingBufferStatus.BufferCapacity) * RingBufferConfiguration.ByteCountOfDataObj;
    ReadAddr := pBufferStart + RingBufferConfiguration.ReadByteOffset;

    // Step 3: Read memory
    SUPER^.RingBufferStatus.CountBytesRead := Tc2_System.MEMMOVE(
        srcAddr := ReadAddr,
        destAddr := ADR(LastObjRead),
        n := RingBufferConfiguration.ByteCountOfDataObj
    );

    // Step 4: Handle result
    IF SUPER^.RingBufferStatus.CountBytesRead = RingBufferConfiguration.ByteCountOfDataObj THEN
        RingBufferStatus.ObjectWasReadPrimary := TRUE;

        RemoveIncrement := RemoveIncrement + 1;

        // Update index and pRemove based on RemoveIncrement
        RemoveIndex := (RemoveIncrement MOD RingBufferStatus.BufferCapacity)
                       + GPL_RingBuffer.MIN_LOGENTRIES;

        pRemove := pBufferStart + 
                   (RemoveIncrement MOD RingBufferStatus.BufferCapacity) * RingBufferConfiguration.ByteCountOfDataObj;

        SUPER^.RingBufferStatus.GlobalCounter := SUPER^.RingBufferStatus.GlobalCounter - 1;
        ReadObject := LastObjRead;  // Return the read object
    ELSE
        RingBufferStatus.ObjectWasReadPrimary := FALSE;
        LastObjRead.Message := ''; // 🛠 Corrected
        Error := TRUE;
    END_IF
ELSE
    RingBufferStatus.ObjectWasReadPrimary := FALSE;
    LastObjRead.Message := ''; // 🛠 Corrected
    Error := TRUE;
END_IF

UpdateObjectCtInBuffers();
END_METHOD

METHOD PUBLIC RemoveObject
VAR_OUTPUT
    Error : BOOL;
END_VAR
VAR
    ByteSize : UDINT;
    Addr     : PVOID;
END_VAR
Error := FALSE;
ByteSize := RingBufferConfiguration.ByteCountOfDataObj;

IF RingBufferStatus.ObjectCountInBufferPrim = 0 THEN   (* nothing to pop *)
    Error := TRUE;
    RETURN;
END_IF;

Addr := pBufferStart +
        (RemoveIncrement MOD RingBufferStatus.BufferCapacity) * ByteSize;

IF Tc2_System.MEMMOVE(srcAddr := Addr, destAddr := ADR(LastObjRemoved), n := ByteSize) <> ByteSize THEN
    Error := TRUE;
    RETURN;
END_IF;
Tc2_System.MEMSET(destAddr := Addr, fillByte := 16#00, n := ByteSize);

(* advance remove side *)
RemoveIncrement := RemoveIncrement + 1;
RemoveIndex     := (RemoveIncrement MOD RingBufferStatus.BufferCapacity)
                 + GPL_RingBuffer.MIN_LOGENTRIES;
pRemove         := pBufferStart +
                   (RemoveIncrement MOD RingBufferStatus.BufferCapacity) * ByteSize;

(* counters / flags *)
RingBufferStatus.ObjectCountInBufferPrim := RingBufferStatus.ObjectCountInBufferPrim - 1;
IF RingBufferStatus.GlobalCounter > 0 THEN
    RingBufferStatus.GlobalCounter := RingBufferStatus.GlobalCounter - 1;
END_IF;

RingBufferStatus.ObjectWasRemovedPrimary := TRUE;

RingBufferStatus.Overwriting  := FALSE;                                 (* we freed space *)
RingBufferStatus.WillOverwrite :=                                     (* preview for next cycle *)
    (RingBufferStatus.ObjectCountInBufferPrim = RingBufferStatus.BufferCapacity);

(* derived *)
RingBufferStatus.BufferIsFullPrim :=
    (RingBufferStatus.ObjectCountInBufferPrim = RingBufferStatus.BufferCapacity);
RingBufferStatus.ByteCountInBufferPrim :=
    RingBufferStatus.ObjectCountInBufferPrim * ByteSize;
END_METHOD

METHOD PROTECTED UpdateRemovePointer
VAR_INPUT
  pRemovePtr  : PVOID;
END_VAR
pRemove := ADR(Buffer[RemoveIndex]);

pRemoveUpdated  := TRUE;
END_METHOD

METHOD PROTECTED UpdateWritePointer
VAR_INPUT
  pWritePtr  : PVOID;
END_VAR
IF (WriteIndex = GPL_RingBuffer.MIN_LOGENTRIES) THEN
  pWrite        := ADR(Buffer[GPL_RingBuffer.MIN_LOGENTRIES]);
ELSIF (WriteIndex > GPL_RingBuffer.MIN_LOGENTRIES) AND
  (WriteIndex <= GPL_RingBuffer.MAX_LOGENTRIES) THEN
  pWrite        := IncrementPointer(pPointer  := pWrite, ByteCtIncrement := RingBufferConfiguration.ByteCountOfDataObj);
END_IF

pWriteUpdated   := TRUE;
END_METHOD

(* Basic component initialization logic*)
METHOD PROTECTED _Initialize : BOOL
VAR
	InterimInit : BOOL;
END_VAR
InterimInit := _InitializeChildrenDependencies();

InterimInit	:= _InitializeReferences();

// IF NOT InterimInit THEN
// 	IF BaseConfiguration.LogTraceConfiguration.What.xLogToEventLogger THEN
// 		TraceWithSeverity(Message := Tc2_Standard.CONCAT('Initialization Failed at ', __POUNAME()), Severity := Global.TcEventSeverity.Error);
// 	END_IF
// END_IF

RingBufferStatus.BufferCapacity  := (GPL_RingBuffer.MAX_LOGENTRIES - GPL_RingBuffer.MIN_LOGENTRIES) +1;

WriteIncrement  := 0;
RemoveIncrement := 0;
WriteIndex      := GPL_RingBuffer.MIN_LOGENTRIES;
RemoveIndex     := GPL_RingBuffer.MIN_LOGENTRIES;
PeekIndex	    := GPL_RingBuffer.MIN_LOGENTRIES;

pBufferStart	:= ADR(Buffer[GPL_RingBuffer.MIN_LOGENTRIES]);

RingBufferConfiguration.ByteCountOfDataObj      := SIZEOF(Buffer[GPL_RingBuffer.MIN_LOGENTRIES]);

IF (pWrite = Tc3_Module.NULL) THEN
  pWrite  := ADR(Buffer[GPL_RingBuffer.MIN_LOGENTRIES]);
END_IF

IF (pRemove = Tc3_Module.NULL) THEN
  pRemove  := ADR(Buffer[GPL_RingBuffer.MIN_LOGENTRIES]);
END_IF

InterimInit	:= _SetDependencyConfiguration();

_Initialize 	:= InterimInit;
END_METHOD

METHOD ClearBuffer
MEMSET(destAddr := ADR(Buffer[GPL_RingBuffer.MIN_LOGENTRIES]), fillByte := 16#00, n := (RingBufferConfiguration.ByteCountOfDataObj*SUPER^.RingBufferStatus.BufferCapacity));

WriteIncrement := 0;
RemoveIncrement := 0;
SUPER^.RingBufferStatus.GlobalCounter := 0;
pWrite := ADR(Buffer[GPL_RingBuffer.MIN_LOGENTRIES]);
pRemove := ADR(Buffer[GPL_RingBuffer.MIN_LOGENTRIES]);
UpdateObjectCtInBuffers();
END_METHOD

PROPERTY P_Buffer : REFERENCE TO ARRAY[GPL_RingBuffer.MIN_LOGENTRIES..GPL_RingBuffer.MAX_LOGENTRIES] OF ST_LogEntry;
GET
P_Buffer REF= Buffer;
END_GET
END_PROPERTY

END_FUNCTION_BLOCK

// RingBuffer/ITFs/I_RingBufferLogEntry
INTERFACE I_RingBufferLogEntry EXTENDS I_RingBufferBase

METHOD PUBLIC AddObject
VAR_INPUT
  RefObject           : REFERENCE TO ST_LogEntry;
END_VAR
VAR_OUTPUT
  Error               : BOOL;
END_VAR
END_METHOD

PROPERTY P_Buffer : REFERENCE TO ARRAY[GPL_RingBuffer.MIN_LOGENTRIES..GPL_RingBuffer.MAX_LOGENTRIES] OF ST_LogEntry;
GET
END_GET
END_PROPERTY

PROPERTY P_LastObjectPeeked : REFERENCE TO ST_LogEntry
GET
END_GET
END_PROPERTY

PROPERTY P_LastObjectRead : REFERENCE TO ST_LogEntry
GET
END_GET
END_PROPERTY

PROPERTY P_LastObjectRemoved : REFERENCE TO ST_LogEntry
GET
END_GET
END_PROPERTY

METHOD PUBLIC PeekObject : ST_LogEntry
END_METHOD

METHOD PUBLIC ReadObject : ST_LogEntry
VAR_OUTPUT
  Error : BOOL;
END_VAR
END_METHOD

END_INTERFACE

// RingBuffer/ITFs/I_RingBufferString
INTERFACE I_RingBufferString EXTENDS I_RingBufferBase

METHOD PUBLIC AddObject
VAR_INPUT
  RefObject           : REFERENCE TO STRING;
END_VAR
VAR_OUTPUT
  Error               : BOOL;
END_VAR
END_METHOD

PROPERTY P_Buffer : REFERENCE TO ARRAY[GPL_RingBuffer.MIN_NUMBER_OBJECTS..GPL_RingBuffer.MAX_NUMBER_OBJECTS] OF STRING;
GET
END_GET
END_PROPERTY

PROPERTY P_LastObjectPeeked : REFERENCE TO STRING
GET
END_GET
END_PROPERTY

PROPERTY P_LastObjectRead : REFERENCE TO STRING
GET
END_GET
END_PROPERTY

PROPERTY P_LastObjectRemoved : REFERENCE TO STRING
GET
END_GET
END_PROPERTY

METHOD PUBLIC PeekObject : STRING
END_METHOD

METHOD PUBLIC ReadObject : STRING
VAR_OUTPUT
  Error : BOOL;
END_VAR
END_METHOD

END_INTERFACE

// RingBuffer/ITFs/I_RingBufferUINT
INTERFACE I_RingBufferUINT EXTENDS I_RingBufferBase

METHOD PUBLIC AddObject
VAR_INPUT
  RefObject           : REFERENCE TO UINT;
END_VAR
VAR_OUTPUT
  Error               : BOOL;
END_VAR
END_METHOD

PROPERTY P_Buffer : REFERENCE TO ARRAY[GPL_RingBuffer.MIN_NUMBER_OBJECTS..GPL_RingBuffer.MAX_NUMBER_OBJECTS] OF UINT;
GET
END_GET
END_PROPERTY

PROPERTY P_LastObjectPeeked : REFERENCE TO UINT
GET
END_GET
END_PROPERTY

PROPERTY P_LastObjectRead : REFERENCE TO UINT
GET
END_GET
END_PROPERTY

PROPERTY P_LastObjectRemoved : REFERENCE TO UINT
GET
END_GET
END_PROPERTY

METHOD PUBLIC PeekObject : UINT
END_METHOD

METHOD PUBLIC ReadObject : UINT
VAR_OUTPUT
  Error : BOOL;
END_VAR
END_METHOD

END_INTERFACE

// RingBuffer/POUs/FB_RingBufferString
{attribute 'no_explicit_call' := 'do not call this POU directly'}
FUNCTION_BLOCK FB_RingBufferString EXTENDS FB_RingBufferBase IMPLEMENTS I_RingBufferBase, I_RingBufferString
VAR
  Buffer              	: ARRAY[GPL_RingBuffer.MIN_NUMBER_OBJECTS..GPL_RingBuffer.MAX_NUMBER_OBJECTS] OF STRING;
  LastObjRemoved		: STRING;
  LastObjPeeked			: STRING;
  LastObjRead			: STRING;
END_VAR

METHOD ClearLastRemoved
MEMSET(destAddr := ADR(LastObjRemoved), fillByte := 16#00, n := RingBufferConfiguration.ByteCountOfDataObj);
END_METHOD

PROPERTY P_RingBufferStatus : REFERENCE TO ST_RingBufferStatus
GET
P_RingBufferStatus REF= SUPER^.RingBufferStatus;
END_GET
END_PROPERTY

METHOD PUBLIC RemoveObject
VAR_OUTPUT
    Error : BOOL;
END_VAR
VAR
    ByteSize : UDINT;
    Addr     : PVOID;
END_VAR
Error := FALSE;
ByteSize := RingBufferConfiguration.ByteCountOfDataObj;

IF RingBufferStatus.ObjectCountInBufferPrim = 0 THEN   (* nothing to pop *)
    Error := TRUE;
    RETURN;
END_IF;

Addr := pBufferStart +
        (RemoveIncrement MOD RingBufferStatus.BufferCapacity) * ByteSize;

IF Tc2_System.MEMMOVE(srcAddr := Addr, destAddr := ADR(LastObjRemoved), n := ByteSize) <> ByteSize THEN
    Error := TRUE;
    RETURN;
END_IF;
Tc2_System.MEMSET(destAddr := Addr, fillByte := 16#00, n := ByteSize);

(* advance remove side *)
RemoveIncrement := RemoveIncrement + 1;
RemoveIndex     := (RemoveIncrement MOD RingBufferStatus.BufferCapacity)
                 + GPL_RingBuffer.MIN_NUMBER_OBJECTS;
pRemove         := pBufferStart +
                   (RemoveIncrement MOD RingBufferStatus.BufferCapacity) * ByteSize;

(* counters / flags *)
RingBufferStatus.ObjectCountInBufferPrim := RingBufferStatus.ObjectCountInBufferPrim - 1;
IF RingBufferStatus.GlobalCounter > 0 THEN
    RingBufferStatus.GlobalCounter := RingBufferStatus.GlobalCounter - 1;
END_IF;

RingBufferStatus.ObjectWasRemovedPrimary := TRUE;

RingBufferStatus.Overwriting  := FALSE;                                 (* we freed space *)
RingBufferStatus.WillOverwrite :=                                     (* preview for next cycle *)
    (RingBufferStatus.ObjectCountInBufferPrim = RingBufferStatus.BufferCapacity);

(* derived *)
RingBufferStatus.BufferIsFullPrim :=
    (RingBufferStatus.ObjectCountInBufferPrim = RingBufferStatus.BufferCapacity);
RingBufferStatus.ByteCountInBufferPrim :=
    RingBufferStatus.ObjectCountInBufferPrim * ByteSize;
END_METHOD

METHOD PUBLIC AddObject
VAR_INPUT
    RefObject : REFERENCE TO STRING;
END_VAR
VAR_OUTPUT
    Error : BOOL;
END_VAR
VAR
    ByteSize   : UDINT;
    ByteOffset : UDINT;
    WriteAddr  : PVOID;
END_VAR
Error := FALSE;
ByteSize := RingBufferConfiguration.ByteCountOfDataObj;

(* ---------- GUARDS ---------- *)
IF (RingBufferStatus.BufferCapacity = 0) OR (NOT __ISVALIDREF(RefObject)) THEN
    Error := TRUE;                           (* zero-capacity or bogus ref *)
    RETURN;
END_IF;
// IF LEN(RefObject) > SIZEOF(RefObject) THEN
//     Error := TRUE;                           (* over-sized payload *)
//     RETURN;
// END_IF;

(* ---------- PREDICT / PREP ---------- *)
RingBufferStatus.WillOverwrite :=
    (RingBufferStatus.ObjectCountInBufferPrim >= RingBufferStatus.BufferCapacity);

ByteOffset := (WriteIncrement MOD RingBufferStatus.BufferCapacity) * ByteSize;
WriteAddr  := pBufferStart + ByteOffset;

(* ---------- WRITE ---------- *)
IF Tc2_System.MEMMOVE(srcAddr := ADR(RefObject), destAddr := WriteAddr, n := ByteSize) <> ByteSize THEN
    Error := TRUE;
    RETURN;
END_IF;

(* ---------- ADVANCE WRITE POINTERS ---------- *)
WriteIncrement := WriteIncrement + 1;
WriteIndex := (WriteIncrement MOD RingBufferStatus.BufferCapacity)
            + GPL_RingBuffer.MIN_NUMBER_OBJECTS;

(* ---------- COUNTERS & FLAGS ---------- *)
IF RingBufferStatus.WillOverwrite THEN
    (* buffer is full – push remove side forward one slot *)
    RemoveIncrement := RemoveIncrement + 1;
    pRemove := pBufferStart
             + (RemoveIncrement MOD RingBufferStatus.BufferCapacity) * ByteSize;
    RingBufferStatus.Overwriting := TRUE;              (* occurred *this* cycle *)
ELSE
    RingBufferStatus.ObjectCountInBufferPrim := RingBufferStatus.ObjectCountInBufferPrim + 1;
    RingBufferStatus.GlobalCounter           := RingBufferStatus.GlobalCounter + 1;
    RingBufferStatus.Overwriting             := FALSE;
END_IF;

RingBufferStatus.ObjectWasAddedPrimary := TRUE;

(* ---------- STATE FOR NEXT SCAN ---------- *)
RingBufferStatus.WillOverwrite :=
    (RingBufferStatus.ObjectCountInBufferPrim >= RingBufferStatus.BufferCapacity);

(* ---------- DERIVED VALUES ---------- *)
RingBufferStatus.BufferIsFullPrim :=
    (RingBufferStatus.ObjectCountInBufferPrim = RingBufferStatus.BufferCapacity);
RingBufferStatus.ByteCountInBufferPrim :=
    RingBufferStatus.ObjectCountInBufferPrim * ByteSize;
END_METHOD

PROPERTY P_LastObjectPeeked : REFERENCE TO STRING
GET
P_LastObjectPeeked REF= LastObjPeeked;
END_GET
END_PROPERTY

PROPERTY P_LastObjectRead : REFERENCE TO STRING
GET
P_LastObjectRead REF= LastObjRead;
END_GET
END_PROPERTY

PROPERTY P_LastObjectRemoved : REFERENCE TO STRING
GET
P_LastObjectRemoved REF= LastObjRemoved;
END_GET
END_PROPERTY

METHOD PUBLIC PeekObject : STRING
PeekIndex := (RemoveIncrement MOD SUPER^.RingBufferStatus.BufferCapacity) + GPL_RingBuffer.MIN_NUMBER_OBJECTS;
PeekAddr := pBufferStart + (PeekIndex - GPL_RingBuffer.MIN_NUMBER_OBJECTS) * RingBufferConfiguration.ByteCountOfDataObj;

// Step 2: Conditional peek (non-mutating)
IF SUPER^.RingBufferStatus.GlobalCounter > 0 THEN
    SUPER^.RingBufferStatus.CountBytesPeeked := Tc2_System.MEMMOVE(
        srcAddr := PeekAddr,
        destAddr := ADR(LastObjPeeked),
        n := RingBufferConfiguration.ByteCountOfDataObj
    );

    IF SUPER^.RingBufferStatus.CountBytesPeeked > 0 THEN
        RingBufferStatus.ObjectWasPeekedPrimary := TRUE;
		PeekObject	:= LastObjPeeked;
    END_IF
ELSE
    RingBufferStatus.ObjectWasPeekedPrimary := FALSE;
    LastObjPeeked := '';
END_IF
END_METHOD

METHOD ReadObject : STRING
VAR_OUTPUT
  Error : BOOL;
END_VAR
// Step 1: Check if buffer has data
IF SUPER^.RingBufferStatus.GlobalCounter > 0 THEN

    // Step 2: Calculate read offset and pointer
    RingBufferConfiguration.ReadByteOffset := (RemoveIncrement MOD RingBufferStatus.BufferCapacity) * RingBufferConfiguration.ByteCountOfDataObj;
    ReadAddr := pBufferStart + RingBufferConfiguration.ReadByteOffset;

    // Step 3: Read memory
    SUPER^.RingBufferStatus.CountBytesRead := Tc2_System.MEMMOVE(
        srcAddr := ReadAddr,
        destAddr := ADR(LastObjRead),
        n := RingBufferConfiguration.ByteCountOfDataObj
    );

    // Step 4: Handle result
    IF SUPER^.RingBufferStatus.CountBytesRead = RingBufferConfiguration.ByteCountOfDataObj THEN
        RingBufferStatus.ObjectWasReadPrimary := TRUE;

        RemoveIncrement := RemoveIncrement + 1;

        // Update index and pRemove based on RemoveIncrement
        RemoveIndex := (RemoveIncrement MOD RingBufferStatus.BufferCapacity)
                       + GPL_RingBuffer.MIN_NUMBER_OBJECTS;

        pRemove := pBufferStart + 
                   (RemoveIncrement MOD RingBufferStatus.BufferCapacity) * RingBufferConfiguration.ByteCountOfDataObj;

        SUPER^.RingBufferStatus.GlobalCounter := SUPER^.RingBufferStatus.GlobalCounter - 1;
    ELSE
        RingBufferStatus.ObjectWasReadPrimary := FALSE;
        LastObjRead := ''; // 🛠 Corrected
        Error := TRUE;
    END_IF
ELSE
    RingBufferStatus.ObjectWasReadPrimary := FALSE;
    LastObjRead := ''; // 🛠 Corrected
    Error := TRUE;
END_IF

UpdateObjectCtInBuffers();
END_METHOD

METHOD PROTECTED UpdateRemovePointer
VAR_INPUT
  pRemovePtr  : PVOID;
END_VAR
pRemove := ADR(Buffer[RemoveIndex]);

pRemoveUpdated  := TRUE;
END_METHOD

METHOD PROTECTED UpdateWritePointer
VAR_INPUT
  pWritePtr  : PVOID;
END_VAR
IF (WriteIndex = GPL_RingBuffer.MIN_NUMBER_OBJECTS) THEN
  pWrite        := ADR(Buffer[GPL_RingBuffer.MIN_NUMBER_OBJECTS]);
ELSIF (WriteIndex > GPL_RingBuffer.MIN_NUMBER_OBJECTS) AND 
  (WriteIndex <= GPL_RingBuffer.MAX_NUMBER_OBJECTS) THEN
  pWrite        := IncrementPointer(pPointer  := pWrite, ByteCtIncrement := RingBufferConfiguration.ByteCountOfDataObj);
END_IF

pWriteUpdated   := TRUE;
END_METHOD

(* Basic component initialization logic*)
METHOD PROTECTED _Initialize : BOOL
VAR
	InterimInit : BOOL;
END_VAR
InterimInit := _InitializeChildrenDependencies();

InterimInit	:= _InitializeReferences();

IF NOT InterimInit THEN
	IF BaseConfiguration.LogTraceConfiguration.What.xLogToEventLogger THEN
		TraceWithSeverity(Message := Tc2_Standard.CONCAT('Initialization Failed at ', __POUNAME()), Severity := Global.TcEventSeverity.Error);
	END_IF
END_IF

RingBufferStatus.BufferCapacity  := (GPL_RingBuffer.MAX_NUMBER_OBJECTS - GPL_RingBuffer.MIN_NUMBER_OBJECTS) +1;

RemoveIndex  := GPL_RingBuffer.MIN_NUMBER_OBJECTS;
PeekIndex	 := GPL_RingBuffer.MIN_NUMBER_OBJECTS;

pBufferStart	:= ADR(Buffer[GPL_RingBuffer.MIN_NUMBER_OBJECTS]);

RingBufferConfiguration.ByteCountOfDataObj      := SIZEOF(Buffer[GPL_RingBuffer.MIN_NUMBER_OBJECTS]);

IF (pWrite = Tc3_Module.NULL) THEN
  pWrite  := ADR(Buffer[GPL_RingBuffer.MIN_NUMBER_OBJECTS]);
END_IF

IF (pRemove = Tc3_Module.NULL) THEN
  pRemove  := ADR(Buffer[GPL_RingBuffer.MIN_NUMBER_OBJECTS]);
END_IF

InterimInit	:= _SetDependencyConfiguration();

_Initialize 	:= InterimInit;
END_METHOD

METHOD ClearBuffer
MEMSET(destAddr := ADR(Buffer[GPL_RingBuffer.MIN_NUMBER_OBJECTS]), fillByte := 16#00, n := (RingBufferConfiguration.ByteCountOfDataObj*SUPER^.RingBufferStatus.BufferCapacity));

WriteIncrement := 0;
RemoveIncrement := 0;
SUPER^.RingBufferStatus.GlobalCounter := 0;
pWrite := ADR(Buffer[GPL_RingBuffer.MIN_NUMBER_OBJECTS]);
pRemove := ADR(Buffer[GPL_RingBuffer.MIN_NUMBER_OBJECTS]);
UpdateObjectCtInBuffers();
END_METHOD

PROPERTY P_Buffer : REFERENCE TO ARRAY[GPL_RingBuffer.MIN_NUMBER_OBJECTS..GPL_RingBuffer.MAX_NUMBER_OBJECTS] OF STRING;
GET
P_Buffer REF= Buffer;
END_GET
END_PROPERTY

END_FUNCTION_BLOCK

// RingBuffer/POUs/FB_RingBufferUINT
{attribute 'no_explicit_call' := 'do not call this POU directly'}
FUNCTION_BLOCK FB_RingBufferUINT EXTENDS FB_RingBufferBase IMPLEMENTS I_RingBufferBase, I_RingBufferUINT
VAR
  Buffer              	: ARRAY[GPL_RingBuffer.MIN_NUMBER_OBJECTS..GPL_RingBuffer.MAX_NUMBER_OBJECTS] OF UINT;
  LastObjRemoved		: UINT;
  LastObjPeeked			: UINT;
  LastObjRead			: UINT;
END_VAR

METHOD ClearLastRemoved
MEMSET(destAddr := ADR(LastObjRemoved), fillByte := 16#00, n := RingBufferConfiguration.ByteCountOfDataObj);
END_METHOD

PROPERTY P_RingBufferStatus : REFERENCE TO ST_RingBufferStatus
GET
P_RingBufferStatus REF= SUPER^.RingBufferStatus;
END_GET
END_PROPERTY

METHOD PUBLIC RemoveObject
VAR_OUTPUT
    Error : BOOL;
END_VAR
VAR
    ByteSize : UDINT;
    Addr     : PVOID;
END_VAR
Error := FALSE;
ByteSize := RingBufferConfiguration.ByteCountOfDataObj;

IF RingBufferStatus.ObjectCountInBufferPrim = 0 THEN   (* nothing to pop *)
    Error := TRUE;
    RETURN;
END_IF;

Addr := pBufferStart +
        (RemoveIncrement MOD RingBufferStatus.BufferCapacity) * ByteSize;

IF Tc2_System.MEMMOVE(srcAddr := Addr, destAddr := ADR(LastObjRemoved), n := ByteSize) <> ByteSize THEN
    Error := TRUE;
    RETURN;
END_IF;
Tc2_System.MEMSET(destAddr := Addr, fillByte := 16#00, n := ByteSize);

(* advance remove side *)
RemoveIncrement := RemoveIncrement + 1;
RemoveIndex     := (RemoveIncrement MOD RingBufferStatus.BufferCapacity)
                 + GPL_RingBuffer.MIN_NUMBER_OBJECTS;
pRemove         := pBufferStart +
                   (RemoveIncrement MOD RingBufferStatus.BufferCapacity) * ByteSize;

(* counters / flags *)
RingBufferStatus.ObjectCountInBufferPrim := RingBufferStatus.ObjectCountInBufferPrim - 1;
IF RingBufferStatus.GlobalCounter > 0 THEN
    RingBufferStatus.GlobalCounter := RingBufferStatus.GlobalCounter - 1;
END_IF;

RingBufferStatus.ObjectWasRemovedPrimary := TRUE;

RingBufferStatus.Overwriting  := FALSE;                                 (* we freed space *)
RingBufferStatus.WillOverwrite :=                                     (* preview for next cycle *)
    (RingBufferStatus.ObjectCountInBufferPrim = RingBufferStatus.BufferCapacity);

(* derived *)
RingBufferStatus.BufferIsFullPrim :=
    (RingBufferStatus.ObjectCountInBufferPrim = RingBufferStatus.BufferCapacity);
RingBufferStatus.ByteCountInBufferPrim :=
    RingBufferStatus.ObjectCountInBufferPrim * ByteSize;
END_METHOD

METHOD PUBLIC AddObject
VAR_INPUT
    RefObject : REFERENCE TO UINT;
END_VAR
VAR_OUTPUT
    Error : BOOL;
END_VAR
VAR
    ByteSize   : UDINT;
    ByteOffset : UDINT;
    WriteAddr  : PVOID;
END_VAR
//Uncomment - will generate and put random numbers into the Ring Buffer
//Random(Num => randLreal); // Do not provide Seed for runtime randomness
//RefObject := LREAL_TO_UINT(randLreal * UINT#65535); // scale to 0..65534

Error := FALSE;
ByteSize := RingBufferConfiguration.ByteCountOfDataObj;

(* ---------- GUARDS ---------- *)
IF (RingBufferStatus.BufferCapacity = 0) OR (NOT __ISVALIDREF(RefObject)) THEN
    Error := TRUE;                           (* zero-capacity or bogus ref *)
    RETURN;
END_IF;
// IF LEN(RefObject) > SIZEOF(RefObject) THEN
//     Error := TRUE;                           (* over-sized payload *)
//     RETURN;
// END_IF;

(* ---------- PREDICT / PREP ---------- *)
RingBufferStatus.WillOverwrite :=
    (RingBufferStatus.ObjectCountInBufferPrim >= RingBufferStatus.BufferCapacity);

ByteOffset := (WriteIncrement MOD RingBufferStatus.BufferCapacity) * ByteSize;
WriteAddr  := pBufferStart + ByteOffset;

(* ---------- WRITE ---------- *)
IF Tc2_System.MEMMOVE(srcAddr := ADR(RefObject), destAddr := WriteAddr, n := ByteSize) <> ByteSize THEN
    Error := TRUE;
    RETURN;
END_IF;

(* ---------- ADVANCE WRITE POINTERS ---------- *)
WriteIncrement := WriteIncrement + 1;
WriteIndex := (WriteIncrement MOD RingBufferStatus.BufferCapacity)
            + GPL_RingBuffer.MIN_NUMBER_OBJECTS;

(* ---------- COUNTERS & FLAGS ---------- *)
IF RingBufferStatus.WillOverwrite THEN
    (* buffer is full – push remove side forward one slot *)
    RemoveIncrement := RemoveIncrement + 1;
    pRemove := pBufferStart
             + (RemoveIncrement MOD RingBufferStatus.BufferCapacity) * ByteSize;
    RingBufferStatus.Overwriting := TRUE;              (* occurred *this* cycle *)
ELSE
    RingBufferStatus.ObjectCountInBufferPrim := RingBufferStatus.ObjectCountInBufferPrim + 1;
    RingBufferStatus.GlobalCounter           := RingBufferStatus.GlobalCounter + 1;
    RingBufferStatus.Overwriting             := FALSE;
END_IF;

RingBufferStatus.ObjectWasAddedPrimary := TRUE;

(* ---------- STATE FOR NEXT SCAN ---------- *)
RingBufferStatus.WillOverwrite :=
    (RingBufferStatus.ObjectCountInBufferPrim >= RingBufferStatus.BufferCapacity);

(* ---------- DERIVED VALUES ---------- *)
RingBufferStatus.BufferIsFullPrim :=
    (RingBufferStatus.ObjectCountInBufferPrim = RingBufferStatus.BufferCapacity);
RingBufferStatus.ByteCountInBufferPrim :=
    RingBufferStatus.ObjectCountInBufferPrim * ByteSize;
END_METHOD

PROPERTY P_LastObjectPeeked : REFERENCE TO UINT
GET
P_LastObjectPeeked REF= LastObjPeeked;
END_GET
END_PROPERTY

PROPERTY P_LastObjectRead : REFERENCE TO UINT
GET
P_LastObjectRead REF= LastObjRead;
END_GET
END_PROPERTY

PROPERTY P_LastObjectRemoved : REFERENCE TO UINT
GET
P_LastObjectRemoved REF= LastObjRemoved;
END_GET
END_PROPERTY

METHOD PUBLIC PeekObject : UINT
PeekIndex := (RemoveIncrement MOD SUPER^.RingBufferStatus.BufferCapacity) + GPL_RingBuffer.MIN_NUMBER_OBJECTS;
PeekAddr := pBufferStart + (PeekIndex - GPL_RingBuffer.MIN_NUMBER_OBJECTS) * RingBufferConfiguration.ByteCountOfDataObj;

// Step 2: Conditional peek (non-mutating)
IF SUPER^.RingBufferStatus.GlobalCounter > 0 THEN
    SUPER^.RingBufferStatus.CountBytesPeeked := Tc2_System.MEMMOVE(
        srcAddr := PeekAddr,
        destAddr := ADR(LastObjPeeked),
        n := RingBufferConfiguration.ByteCountOfDataObj
    );

    IF SUPER^.RingBufferStatus.CountBytesPeeked > 0 THEN
        RingBufferStatus.ObjectWasPeekedPrimary := TRUE;
		PeekObject	:= LastObjPeeked;
    END_IF
ELSE
    RingBufferStatus.ObjectWasPeekedPrimary := FALSE;
    LastObjPeeked := 0;
END_IF
END_METHOD

METHOD ReadObject : UINT
VAR_OUTPUT
  Error : BOOL;
END_VAR
// Step 1: Check if buffer has data
IF SUPER^.RingBufferStatus.GlobalCounter > 0 THEN

    // Step 2: Calculate read offset and pointer
    RingBufferConfiguration.ReadByteOffset := (RemoveIncrement MOD RingBufferStatus.BufferCapacity) * RingBufferConfiguration.ByteCountOfDataObj;
    ReadAddr := pBufferStart + RingBufferConfiguration.ReadByteOffset;

    // Step 3: Read memory
    SUPER^.RingBufferStatus.CountBytesRead := Tc2_System.MEMMOVE(
        srcAddr := ReadAddr,
        destAddr := ADR(LastObjRead),
        n := RingBufferConfiguration.ByteCountOfDataObj
    );

    // Step 4: Handle result
    IF SUPER^.RingBufferStatus.CountBytesRead = RingBufferConfiguration.ByteCountOfDataObj THEN
        RingBufferStatus.ObjectWasReadPrimary := TRUE;

        RemoveIncrement := RemoveIncrement + 1;

        // Update index and pRemove based on RemoveIncrement
        RemoveIndex := (RemoveIncrement MOD RingBufferStatus.BufferCapacity)
                       + GPL_RingBuffer.MIN_NUMBER_OBJECTS;

        pRemove := pBufferStart + 
                   (RemoveIncrement MOD RingBufferStatus.BufferCapacity) * RingBufferConfiguration.ByteCountOfDataObj;

        SUPER^.RingBufferStatus.GlobalCounter := SUPER^.RingBufferStatus.GlobalCounter - 1;
    ELSE
        RingBufferStatus.ObjectWasReadPrimary := FALSE;
        LastObjRead := 0;
        Error := TRUE;
    END_IF
ELSE
    RingBufferStatus.ObjectWasReadPrimary := FALSE;
    LastObjRead := 0;
    Error := TRUE;
END_IF

UpdateObjectCtInBuffers();
END_METHOD

METHOD PROTECTED UpdateRemovePointer
VAR_INPUT
  pRemovePtr  : PVOID;
END_VAR
pRemove := ADR(Buffer[RemoveIndex]);

pRemoveUpdated  := TRUE;
END_METHOD

METHOD PROTECTED UpdateWritePointer
VAR_INPUT
  pWritePtr  : PVOID;
END_VAR
IF (WriteIndex = GPL_RingBuffer.MIN_NUMBER_OBJECTS) THEN
  pWrite        := ADR(Buffer[GPL_RingBuffer.MIN_NUMBER_OBJECTS]);
ELSIF (WriteIndex > GPL_RingBuffer.MIN_NUMBER_OBJECTS) AND 
  (WriteIndex <= GPL_RingBuffer.MAX_NUMBER_OBJECTS) THEN
  pWrite        := IncrementPointer(pPointer  := pWrite, ByteCtIncrement := RingBufferConfiguration.ByteCountOfDataObj);
END_IF

pWriteUpdated   := TRUE;
END_METHOD

(* Basic component initialization logic*)
METHOD PROTECTED _Initialize : BOOL
VAR
	InterimInit : BOOL;
END_VAR
InterimInit := _InitializeChildrenDependencies();

InterimInit	:= _InitializeReferences();

IF NOT InterimInit THEN
	IF BaseConfiguration.LogTraceConfiguration.What.xLogToEventLogger THEN
		TraceWithSeverity(Message := Tc2_Standard.CONCAT('Initialization Failed at ', __POUNAME()), Severity := Global.TcEventSeverity.Error);
	END_IF
END_IF

RingBufferStatus.BufferCapacity  := (GPL_RingBuffer.MAX_NUMBER_OBJECTS - GPL_RingBuffer.MIN_NUMBER_OBJECTS) +1;

RemoveIndex  := GPL_RingBuffer.MIN_NUMBER_OBJECTS;
PeekIndex	 := GPL_RingBuffer.MIN_NUMBER_OBJECTS;

pBufferStart	:= ADR(Buffer[GPL_RingBuffer.MIN_NUMBER_OBJECTS]);

RingBufferConfiguration.ByteCountOfDataObj      := SIZEOF(Buffer[GPL_RingBuffer.MIN_NUMBER_OBJECTS]);

IF (pWrite = Tc3_Module.NULL) THEN
  pWrite  := ADR(Buffer[GPL_RingBuffer.MIN_NUMBER_OBJECTS]);
END_IF

IF (pRemove = Tc3_Module.NULL) THEN
  pRemove  := ADR(Buffer[GPL_RingBuffer.MIN_NUMBER_OBJECTS]);
END_IF

InterimInit	:= _SetDependencyConfiguration();

_Initialize 	:= InterimInit;
END_METHOD

METHOD ClearBuffer
MEMSET(destAddr := ADR(Buffer[GPL_RingBuffer.MIN_NUMBER_OBJECTS]), fillByte := 16#00, n := (RingBufferConfiguration.ByteCountOfDataObj*SUPER^.RingBufferStatus.BufferCapacity));

WriteIncrement := 0;
RemoveIncrement := 0;
SUPER^.RingBufferStatus.GlobalCounter := 0;
pWrite := ADR(Buffer[GPL_RingBuffer.MIN_NUMBER_OBJECTS]);
pRemove := ADR(Buffer[GPL_RingBuffer.MIN_NUMBER_OBJECTS]);
UpdateObjectCtInBuffers();
END_METHOD

PROPERTY P_Buffer : REFERENCE TO ARRAY[GPL_RingBuffer.MIN_NUMBER_OBJECTS..GPL_RingBuffer.MAX_NUMBER_OBJECTS] OF UINT;
GET
P_Buffer REF= Buffer;
END_GET
END_PROPERTY

END_FUNCTION_BLOCK

// Safety/FB_SafetyDevice
{attribute 'no_explicit_call' := 'do not call this POU directly'}
FUNCTION_BLOCK FB_SafetyDevice EXTENDS FB_BaseCyclic
VAR
	EStopFBErr		AT %I*	: BOOL;
	EDMErr1			AT %I* 	: BOOL;
END_VAR

METHOD CyclicLogic
SUPER^.CyclicLogic();
END_METHOD

END_FUNCTION_BLOCK

// Safety/FB_SafetyGroup
{attribute 'no_explicit_call' := 'do not call this POU directly'}
FUNCTION_BLOCK FB_SafetyGroup EXTENDS FB_BaseCyclic
VAR
	Configuration	: ST_SafetyGroupConfiguration;
	Status			: ST_SafetyGroupStatus;
END_VAR

METHOD PROTECTED _InitializeReferences : BOOL
//Order is important!
BaseConfiguration.InstancePath 	REF= InstancePath;

IF BaseConfiguration.LogTraceConfiguration.When = E_LogTraceWhen.xRunOnInitOnly AND_THEN
   BaseConfiguration.LogTraceConfiguration.What.xLogToEventLogger THEN
	TraceWithSeverity(Message := Tc2_Standard.CONCAT('If you created new data structures, they may not have valid pointer references; Check ', __POUNAME()), Severity := Global.TcEventSeverity.Warning);
END_IF

Configuration.BaseConfiguration		REF= SUPER^.BaseConfiguration;

Status.BaseStatus				REF= SUPER^.BaseStatus;

_InitializeReferences 			:= TRUE; // apply at end of all reference initialization
END_METHOD

METHOD CyclicLogic
SUPER^.CyclicLogic();
END_METHOD

PROPERTY P_SafetyGroupConfiguration : REFERENCE TO ST_SafetyGroupConfiguration
GET
P_SafetyGroupConfiguration REF= Configuration;
END_GET
END_PROPERTY

PROPERTY P_SafetyGroupStatus : REFERENCE TO ST_SafetyGroupStatus
GET
P_SafetyGroupStatus REF= Status;
END_GET
END_PROPERTY

METHOD Reset
VAR_INPUT
	Trig	: BOOL;
END_VAR
Configuration.ErrAck := Trig;
END_METHOD

END_FUNCTION_BLOCK

// Tests/TestFunctions/ThenAssertState
FUNCTION ThenAssertState : BOOL
VAR_INPUT
	testIndex : DINT;
END_VAR
VAR_IN_OUT
	expectedState 		: E_CommandState;
	TestCommand 		: ARRAY[*] OF FB_CommandUnderTest;
	iTestCommand 		: I_CommandUnderTest;
END_VAR

// Validate test index range
IF testIndex < GC_Test.INDEX_TestFB_Command_MIN OR testIndex > GC_Test.INDEX_TestFB_Command_MAX THEN
    ThenAssertState := FALSE;
    RETURN;
END_IF

// Ensure interfaces are available
IF NOT __QUERYINTERFACE(TestCommand[testIndex], iTestCommand) THEN
    ThenAssertState := FALSE;
    RETURN;
END_IF

// Assert the expected state
TcUnit.AssertEquals_UDINT(
    Expected := expectedState,
    Actual := iTestCommand.P_CommandStatus.StepState,
    Message := Tc2_Standard.CONCAT('Expected state: ', TO_STRING(expectedState))
);

ThenAssertState := TRUE;

END_FUNCTION

// Tests/TestFunctions/WhenExecuteCommand
FUNCTION WhenExecuteCommand : BOOL
VAR_INPUT
	testIndex : DINT;
END_VAR
VAR_IN_OUT
	TestCommand 			: ARRAY[*] OF FB_CommandUnderTest;
	TestComponent 			: ARRAY[*] OF FB_ComponentDerivative;
	TestCommandConfig 		: ARRAY[*] OF FB_CmdPermIntlkConfiguration;
	iTestCommand 			: I_CommandUnderTest;
	iTestCommandConfig 		: I_CommandConfiguration;
	iTestComponent 			: I_ComponentFull;
	iTestPermIntlkConfig 	: I_PermIntlkConfiguration;
END_VAR

// Validate test index range and that command is ready
IF testIndex < GC_Test.INDEX_TestFB_Command_MIN OR testIndex > GC_Test.INDEX_TestFB_Command_MAX THEN
    WhenExecuteCommand := FALSE;
    RETURN;
END_IF

// Ensure interfaces are available
IF NOT __QUERYINTERFACE(TestCommand[testIndex], iTestCommand) THEN
    WhenExecuteCommand := FALSE;
    RETURN;
END_IF

// Verify command has been properly configured before execution
IF iTestCommand.P_CommandStatus.ConfigRef.CommandDescription = '' THEN
    // Command might not be configured yet - try to set up basic configuration
    IF __QUERYINTERFACE(TestCommandConfig[testIndex], iTestCommandConfig) THEN
        IF __QUERYINTERFACE(TestComponent[testIndex], iTestComponent) THEN
            IF __QUERYINTERFACE(TestCommandConfig[testIndex], iTestPermIntlkConfig) THEN
                // Basic configuration setup
                iTestCommandConfig.P_CommandConfiguration.CommandDescription := 'Test Command Execution';
                IF __ISVALIDREF(iTestCommandConfig.P_CommandConfiguration.BaseConfiguration) THEN
                    iTestCommandConfig.P_CommandConfiguration.BaseConfiguration.LogTraceConfiguration.When := E_LogTraceWhen.xRunOnInitOnly;
                END_IF
                
                // Inject configurations if not already done
                iTestCommand.InjectConfigurations(
                    iComponent := iTestComponent,
                    iCommandConfiguration := iTestCommandConfig,
                    iPermIntlkConfiguration := iTestPermIntlkConfig
                );
            END_IF
        END_IF
    END_IF
END_IF

// Execute the command
iTestCommand.Execute();

WhenExecuteCommand := TRUE;

END_FUNCTION

// Tests/FB_FileHandlerCsvTests
FUNCTION_BLOCK FB_FileHandlerCsvTests EXTENDS TcUnit.FB_TestSuite
VAR
    FileHandlerCsv : FB_FileHandlerCsv;
    MockCommandConfig : FB_CommandConfiguration;
    iMockCommandConfig : I_CommandConfiguration;
    MockPermIntlkConfig : FB_PermIntlkConfiguration;
    iMockPermIntlkConfig : I_PermIntlkConfiguration;
END_VAR

TEST_CloseFileCommandDispatch();

METHOD TEST_CloseFileCommandDispatch
VAR
    ExpectedPOUName : STRING := 'CloseFile';
    ExpectedCommandIndex : DINT;
    ActualMethodDispatch : DINT;
    ActualLastCommandMessage : STRING;
END_VAR
// Setup - Initialize FileHandlerCsv
FileHandlerCsv.Initialize();

// Setup mock command configuration for CloseFile
iMockCommandConfig := MockCommandConfig;
MockCommandConfig.InjectConfiguration(
    CommandPOUName := 'CloseFile',
    CommandIndex := GC_FILE.INDEX_CLOSEFILE,
    Priority := 1,
    TimeoutTime := T#5S
);

// Setup mock permissive/interlock configuration
iMockPermIntlkConfig := MockPermIntlkConfig;
MockPermIntlkConfig.Initialize();

// Inject configurations into FileHandlerCsv
FileHandlerCsv.InjectCommandConfiguration(
    CmdIndex := GC_FILE.INDEX_CLOSEFILE,
    CommandConfig := iMockCommandConfig
);

FileHandlerCsv.InjectPermIntlkConfiguration(
    CmdIndex := GC_FILE.INDEX_CLOSEFILE,
    PermIntlkConfig := iMockPermIntlkConfig
);

// Force initialization to build hash tables
FileHandlerCsv._Initialize();

// Test: Call CloseFile business logic method
FileHandlerCsv.CloseFile();

// Verify: Check that POUName was extracted correctly
ActualLastCommandMessage := FileHandlerCsv.P_ComponentStatus.LastCommandStatus.LastCommandMessage;
AssertEquals_STRING(
    Expected := ExpectedPOUName,
    Actual := ActualLastCommandMessage,
    Message := 'POUName extraction failed'
);

// Verify: Check that MethodDispatch was set to correct index
ExpectedCommandIndex := GC_FILE.INDEX_CLOSEFILE;
ActualMethodDispatch := FileHandlerCsv.P_ComponentStatus.MethodDispatch;
AssertEquals_DINT(
    Expected := ExpectedCommandIndex,
    Actual := ActualMethodDispatch,
    Message := 'MethodDispatch not set to correct command index'
);

// Test: Verify GetIndexByPOUName works correctly
ActualMethodDispatch := FileHandlerCsv.GetIndexByPOUName(NameIn := 'CloseFile');
AssertEquals_DINT(
    Expected := ExpectedCommandIndex,
    Actual := ActualMethodDispatch,
    Message := 'GetIndexByPOUName failed to find CloseFile command'
);
END_METHOD

END_FUNCTION_BLOCK

// Tests/FB_InterfaceResolutionTests
FUNCTION_BLOCK FB_InterfaceResolutionTests EXTENDS TcUnit.FB_TestSuite
VAR
	TrigIndex							: DINT;
	ActuatorCmdConfiguration			: ARRAY[GC_Actuator.INDEX_COMMAND_MIN..GC_Actuator.INDEX_COMMAND_MAX] OF FB_CmdPermIntlkConfiguration;
	iCommandConfiguration				: ARRAY[GC_Actuator.INDEX_COMMAND_MIN..GC_Actuator.INDEX_COMMAND_MAX] OF I_CommandConfiguration;
	iPermIntlkConfigurationActuator		: ARRAY[GC_Actuator.INDEX_COMMAND_MIN..GC_Actuator.INDEX_COMMAND_MAX] OF I_PermIntlkConfiguration;
	iPermIntlkConfigurationDummy	 	: I_PermIntlkConfiguration;
	ControlModeCmdConfiguration			: ARRAY[GC_ControlMode.INDEX_COMMAND_MIN..GC_ControlMode.INDEX_COMMAND_MAX] OF I_CommandConfiguration;
	ControlModePermIntlkConfiguration	: ARRAY[GC_ControlMode.INDEX_COMMAND_MIN..GC_ControlMode.INDEX_COMMAND_MAX] OF I_PermIntlkConfiguration;
	PermIntlk							: FB_PermIntlk;
	iPermIntlk							: I_PermIntlk := PermIntlk;
	iControlModeTop						: I_ControlMode;
	ControlMode							: FB_ControlMode;
	iControlMode						: I_ControlMode := ControlMode;
	TestActuator 						: FB_Actuator;
END_VAR

GivenActuatorWithInjectedInterfacesExpectAllInterfacesValid();
GivenCommandStatusExpectAllResolvedOrInjected();

METHOD PRIVATE GivenActuatorWithInjectedInterfacesExpectAllInterfacesValid
VAR
	idxCmd                             	: DINT;
	idxPermIntlk                        : DINT;
	AllCommandInterfacesValid       	: BOOL := TRUE;
	AllPermIntlkInterfacesValid     	: BOOL := TRUE;
	SystemPermIntlkIsValid          	: BOOL;
	ControlModeIsValid              	: BOOL;
END_VAR
TEST(__POUNAME());

// Initialization (if needed)
TestActuator.Initialize();

// Check array-based interface injection
FOR idxCmd := GC_Actuator.INDEX_COMMAND_MIN TO GC_Actuator.INDEX_COMMAND_MAX DO
	IF TestActuator.P_TP_CmdConfigurations[idxCmd] = 0 THEN
		AllCommandInterfacesValid := FALSE;
		EXIT;
	END_IF
END_FOR

// Check array-based interface injection
FOR idxPermIntlk := GC_Actuator.INDEX_COMMAND_MIN TO GC_Actuator.INDEX_COMMAND_MAX DO
	IF TestActuator.P_TP_PermIntlkConfigurations[idxPermIntlk] = 0 THEN
		AllPermIntlkInterfacesValid := FALSE;
		EXIT;
	END_IF
END_FOR

// Check single external dependencies
SystemPermIntlkIsValid := (TestActuator.P_TP_iSystemPermIntlk <> 0);
ControlModeIsValid := (TestActuator.P_TP_iControlMode <> 0);

// Assertions
AssertEquals_BOOL(Actual := AllCommandInterfacesValid, Expected := TRUE,
	Message := 'Expected all _iCommandConfiguration entries to be valid (nonzero)');
AssertEquals_BOOL(Actual := AllPermIntlkInterfacesValid, Expected := TRUE,
	Message := 'Expected all _iPermIntlkConfiguration entries to be valid (nonzero)');

AssertEquals_BOOL(Actual := SystemPermIntlkIsValid, Expected := TRUE,
	Message := 'Expected _SystemPermIntlk interface to be valid (nonzero)');
AssertEquals_BOOL(Actual := ControlModeIsValid, Expected := TRUE,
	Message := 'Expected _ControlMode interface to be valid (nonzero)');

TEST_FINISHED();
END_METHOD

METHOD GivenCommandStatusExpectAllResolvedOrInjected
VAR
	idx                             : DINT;
	AllStatusesValid                : BOOL := TRUE;
	ConfigRes                       : E_ConfigurationResolution;
END_VAR
TEST(__POUNAME());

// Simulate initialization if needed
TestActuator.Initialize();

// Evaluate each command status
FOR idx := GC_Actuator.INDEX_COMMAND_MIN TO GC_Actuator.INDEX_COMMAND_MAX DO
	ConfigRes := TestActuator.P_TP_Commands[idx].CommandStatus.CmdConfigurationResolution;

	IF ConfigRes = E_ConfigurationResolution.Local THEN
		AllStatusesValid := FALSE;
		EXIT;
	END_IF
END_FOR

// Assert
AssertEquals_BOOL(Actual := AllStatusesValid, Expected := TRUE,
	Message := 'Expected all command statuses to be resolved via InjectedInterface (no Local)');

TEST_FINISHED();
END_METHOD

METHOD FB_Init : BOOL
VAR_INPUT
	(* if TRUE, the retain variables are initialized (warm start / cold start)*)
	bInitRetains	: BOOL;
	(* if TRUE, the instance afterwards gets moved into the copy code (online change)*)
	bInCopyCode	: BOOL;
END_VAR
FOR TrigIndex := GC_Actuator.INDEX_COMMAND_MIN TO GC_Actuator.INDEX_COMMAND_MAX DO
    iCommandConfiguration[TrigIndex]       := ActuatorCmdConfiguration[TrigIndex]; // implements I_CommandConfiguration
    iPermIntlkConfigurationActuator[TrigIndex] := ActuatorCmdConfiguration[TrigIndex]; // implements I_PermIntlkConfiguration
	
	iCommandConfiguration[TrigIndex].P_CommandConfiguration.CommandIndex			:= TrigIndex;
END_FOR

// TestActuator.InjectActuatorCmdPermIntlkConfigurations(ControlMode := iControlMode, SystemPermIntlk := iPermIntlk, CommandConfigurations := iCommandConfiguration, PermIntlkConfigurations := iPermIntlkConfigurationActuator);

FB_Init := TRUE;
END_METHOD

END_FUNCTION_BLOCK
